(* PLC project services, CODESYS STW CODESYS V3.5 SP11 - ESX-3CS *)
(* stored: creationDateTime 2026-05-19T11:35:05.3616724, version 0.1, modificationDateTime 2026-02-03T11:13:35, organization Isoloader *)

TYPE t_bms_charge_state : (cBMSChargeStateShutdown := 0, cBMSChargeStateDC := 1, cBMSChargeStateAC := 2, cBMSChargeStateOther := 3);
END_TYPE

TYPE t_bms_fault_level : (cBMSFaultLevelNone := 0, cBMSFaultLevelLow := 1, cBMSFaultLevelMedium := 2, cBMSFaultLevelSevere := 3);
END_TYPE

TYPE t_bms_state : (cBMSStateShutdown := 0, cBMSStateStandby := 1, cBMSStateDisconnected := 2, cBMSStateConnected := 3);
END_TYPE

TYPE t_tms_state : (cTMSStateShutdown := 0, cTMSStateCooling := 1, cTMSStateHeating := 2, cTMSStateCirculation := 3);
END_TYPE

TYPE t_charger_diagnostic : (cChargingDiagnostic := 0, cChargingDiagnosticNotOperational := 1, cChargingDiagnosticDisconnected := 2, cChargingDiagnosticConnectedError := 3, cChargingDiagnosticConnectedStandby := 4, cChargingDiagnosticNotInChargingState := 5, cChargingDiagnosticTargetSOCReached := 6, cChargingDiagnosticBMSShutdown := 7, cChargingDiagnosticConnected := 8, cChargingDiagnosticConnectedCharging := 9);
END_TYPE

TYPE t_obc_state : (cOBCStateDisconnected := 0, cOBCStateCharging := 1, cOBCStateStandby := 2, cOBCStateError := 3);
END_TYPE

TYPE t_obc_status : (cOBCStatusNone := 0, cOBCStatusCharging := 1, cOBCStatusStandby := 2, cOBCStatusError := 3);
END_TYPE

TYPE t_active_state : (cActiveStateNone := 0, cActiveStatePre := 1, cActiveStatePost := 2, cActiveStateActive := 3);
END_TYPE

TYPE t_adjust_state : (cAdjustStateNone := 0, cAdjustStateGood := 1, cAdjustStateAdjusting := 2, cAdjustStateError := 3);
END_TYPE

(* {attribute 'qualified_only'} *)
TYPE t_channel_state : (cChannelStateNone := 0, cChannelStateError := 1, cChannelStateOverflow := 2, cChannelStateHeartbeat := 3, cChannelStateEmergency := 4, cChannelStateStarting := 5, cChannelStateReady := 6, cChannelStateGood := 7);
END_TYPE

(* {attribute 'qualified_only'} *)
TYPE t_controller_status : (cControllerStatusNone := 0, cControllerStatusFault := 1, cControllerStatusNotReady := 2, cControllerStatusOnline := 3, cControllerStatusWarning := 4, cControllerStatusReady := 5, cControllerStatusOperating := 6);
END_TYPE

TYPE t_data_type : (cDataTypeNone := 0, cDataTypeEnum := 1, cDataTypeString := 2, cDataTypeUSINT := 3, cDataTypeUINT := 4, cDataTypeULINT := 5, cDataTypeUDINT := 6, cDataTypeINT := 7, cDataTypePercentage := 8, cDataTypeReal := 9, cDataTypeDWORD := 10, cDataTypeBool := 11);
END_TYPE

TYPE t_debug_mask : (cDebugNone := 16#0, cDebugWaitForLog := 16#1, cDebugEnableFailSafeOnCrash := 16#2, cDebugDisableWatchdog := 16#4, cDebugSimulateCrash := 16#100, cDebugSimulateA := 16#200, cDebugSimulateB := 16#400, cDebugSimulateC := 16#800);
END_TYPE

TYPE t_enum_type : (cEnumTypeNone := 0, cEnumTypeActiveState := 1, cEnumTypeAdjustState := 2, cEnumTypeChannelState := 3, cEnumTypeControllerStatus := 4, cEnumTypeDebugMask := 5, cEnumTypeEventCode := 6, cEnumTypeFunctionalMode := 7, cEnumTypeInputMode := 8, cEnumTypeInterlockState := 9, cEnumTypeLedCode := 10, cEnumTypeLockState := 11, cEnumTypeOperatingMethod := 12, cEnumTypeProgMovCode := 13, cEnumTypeProgMovState := 14, cEnumTypeReadyState := 15, cEnumTypeRunState := 16, cEnumTypeShutdownCode := 17, cEnumTypeSpreaderExtensionMethod := 18, cEnumTypeSpreaderExtensionState := 19, cEnumTypeStateCode := 20, cEnumTypeSteerMode := 21, cEnumTypeSubsystem := 22, cEnumTypeSystemMethod := 23, cEnumTypeSystemState := 24, cEnumTypeTopbeamsState := 25, cEnumTypeUiEventCode := 26, cEnumTypeUiId := 27, cEnumTypeUiMode := 28, cEnumTypeUiOrientation := 29, cEnumTypeBMSChargeState := 30, cEnumTypeBMSFaultLevel := 31, cEnumTypeBMSState := 32, cEnumTypeChannelMask := 33, cEnumTypeOBCState := 34, cEnumTypeOBCStatus := 35, cEnumTypeTMSState := 36, cEnumTypeTokenType := 37, cEnumTypeSystemControl := 38, cEnumTypeSeverity := 39, cEnumTypeChargeQualifier := 40, cEnumTypeExecuteOption := 41, cEnumTypeExecuteReturn := 42, cEnumTypeValueStyle := 43, cEnumTypeDataType := 44);
END_TYPE

TYPE t_event_code : (cECNone := 0, cECSystemControl := 1, cECAllowUpState := 2, cECAllowDownState := 3, cECForceMaxState := 4, cECNextState := 5, cECModulation := 6, cECChargeModulation := 8, cECMovementInputInterlock := 9, cECMovementChargeInterlock := 10, cECSecondaryPowerModulation := 11, cECTransitionInitializedStandby := 12, cECTransitionStandbyPreparing := 13, cECTransitionStandbyInitialized := 14, cECTransitionPreparingPreOperational := 15, cECTransitionPreparingCharging := 16, cECTransitionPreparingStandby := 17, cECTransitionChargingPreparing := 18, cECTransitionPreOperationalPreparing := 19, cECTransitionPoweringUpGoOperational := 20, cECTransitionGoOperationalOperational := 21, cECTransitionExitOperationalPoweringDown := 22, cECTransitionPoweringDownPreOperational := 23, cECMetric := 24, cECMax := 63);
END_TYPE

(* {attribute 'qualified_only'} *)
TYPE t_functional_mode : (cFunctionalModeAny := 0, cFunctionalModeDefault := 1, cFunctionalModeTravel := 2, cFunctionalModeLift := 3, cFunctionalModeSpreaderConfiguration := 4, cFunctionalModeTopbeamConfiguration := 5);
END_TYPE

(* {attribute 'qualified_only'} *)
TYPE t_input_mode : (cInputModeNone := 0, cInputModeDefault := 1, cInputModeSpreaderConfiguration := 2, cInputModeTopbeamConfiguration := 3);
END_TYPE

TYPE t_interlock_state : (cInterlockStateNone := 0, cInterlockStateFailure := 1, cInterlockStateError := 2, cInterlockStateErrorNegative := 3, cInterlockStateErrorPositive := 4, cInterlockStateWarning := 5, cInterlockStateOveride := 6, cInterlockStateGood := 7);
END_TYPE

TYPE t_led_code : (cLEDCodeNone := 0, cLEDCodeStartup := 1, cLEDCodeStandby := 2, cLEDCodeNormal := 3, cLEDCodeMaintenance := 4, cLEDCodeSoftwareCrash := 5, cLEDCodeWatchDogDisabled := 6, cLEDCodeFailSafe := 7, cLEDCodeFailSafeSevere := 8);
END_TYPE

(* {attribute 'qualified_only'} *)
TYPE t_lock_state : (cLockStateNone := 0, cLockStateUnlocked := 1, cLockStateLocked := 2, cLockStatePartial := 3);
END_TYPE

(* values of t_machine_state_id: cMSIdSystemState: operating state; cMSIdLocalMessageText: local UIState *)

{attribute 'qualified_only'}
{attribute 'strict'}
TYPE t_machine_state_id : (cMSIdNone := 0, cMSIdSystemState := 1, cMSIdSystemMethodRequest := 2, cMSIdOperatingMode := 3, cMSIdOperatingModeRequest := 4, cMSIdRadioModeResponse := 5, cMSIdMachineHours := 6, cMSIdLightsStatus := 12, cMSIdToggleLightsRequest := 13, cMSIdSpeedModeSlow := 14, cMSIdToggleSpeedModeRequest := 15, cMSIdBatteryLevel := 20, cMSIdMainCurrent := 21, cMSIdChargingCurrent := 22, cMSIdEngineState := 23, cMSIdSteerModeStatus := 30, cMSIdSteerModeRequest := 31, cMSIdSteerModeRequest2WS := 32, cMSIdSteerModeRequest4WS := 33, cMSIdSteerModeRequest4WS90 := 34, cMSIdSteerModeRequestLateral := 35, cMSIdSteerModeRequestCarousel := 36, cMSIdSteerStateA := 37, cMSIdSteerStateB := 38, cMSIdSteerStateC := 39, cMSIdSteerStateD := 40, cMSIdTravelVelocity := 41, cMSIdTravelInterlock := 42, cMSIdTravelInterlockTrace := 43, cMSIdTopbeamABPosition := 44, cMSIdTopbeamCDPosition := 45, cMSIdTopbeamABInterlock := 46, cMSIdTopbeamCDInterlock := 47, cMSIdTopbeamABInterlockTrace := 48, cMSIdTopbeamCDInterlockTrace := 49, cMSIdLiftABPosition := 50, cMSIdLiftCDPosition := 51, cMSIdLiftABInterlock := 52, cMSIdLiftCDInterlock := 53, cMSIdLiftABInterlockTrace := 54, cMSIdLiftCDInterlockTrace := 55, cMSIdLiftTopRequest := 56, cMSIdSpreaderGrabArms := 60, cMSIdToggleSpreaderGrabArmsRequest := 61, cMSIdSpreaderTelescopingExtensionStateRequest6m := 62, cMSIdSpreaderTelescopingExtensionStateRequest9m := 63, cMSIdSpreaderTelescopingExtensionStateRequest12m := 64, cMSIDSpreaderState := 65, cMSIDSpreaderStateA := 66, cMSIDSpreaderStateB := 67, cMSIDSpreaderStateC := 68, cMSIDSpreaderStateD := 69, cMSIDSpreaderLowered := 70, cMSIDSpreaderLoweredA := 71, cMSIDSpreaderLoweredB := 72, cMSIDSpreaderLoweredC := 73, cMSIDSpreaderLoweredD := 74, cMSIdSpreaderTelescopingControl := 75, cMSIdSpreaderGrabArmsDeployControl := 76, cMSIdSpreaderGrabArmsExtendABRequest := 77, cMSIdSpreaderGrabArmsRetractABRequest := 78, cMSIdSpreaderGrabArmsExtendCDRequest := 79, cMSIdSpreaderGrabArmsRetractCDRequest := 80, cMSIdConfigureState := 85, cMSIdConfigureStateValid := 86, cMSIdConfigureMethodRequest := 87, cMSIdReconfigureCheckingRequest := 88, cMSIdUnloadedState := 89, cMSIdLevelState := 90, cMSIdMastsState := 91, cMSIdReconfigureMastsRequest := 92, cMSIdTopbeamsState := 93, cMSIdReconfigureTopbeamsRequest := 94, cMSIdMastAThrottle := 100, cMSIdMastBThrottle := 101, cMSIdMastCThrottle := 102, cMSIdMastDThrottle := 103, cMSIdTopbeamABThrottle := 104, cMSIdTopbeamCDThrottle := 105, cMSIdLocalMessageText := 110, cMSIdLocalMessageDisplayCode := 111, cMSIdLocalStatusText := 112, cMSIdLocalStatusDisplayCode := 113, cMSIdLocalButtonSteerModeSelectEnter := 115, cMSIdLocalButtonSteerModeSelectSwitch := 116, cMSIdLocalButtonSteerModeSelectExit := 117, cMSIDLocalAckMessageEnter := 118, cMSIDLocalAckMessageExit := 119, cMSIDLocalFlashMessageEnter := 120, cMSIDLocalFlashMessageExit := 121, cMSIdLocalButtonConfigureEnter := 122, cMSIdLocalButtonConfigureSwitch := 123, cMSIdLocalButtonConfigureExit := 124, cMSIdLocalButtonMastsSelectEnter := 125, cMSIdLocalButtonMastsSelectSwitch := 126, cMSIdLocalButtonMastsSelectExit := 127, cMSIdLocalButtonTopbeamsSelectEnter := 128, cMSIdLocalButtonTopbeamsSelectSwitch := 129, cMSIdLocalButtonTopbeamsSelectExit := 130, cMSIdLocalButtonUnloadedSelectEnter := 131, cMSIdLocalButtonUnloadedSelectSwitch := 132, cMSIdLocalButtonUnloadedSelectExit := 133, cMSIdLocalButtonLevelSelectEnter := 134, cMSIdLocalButtonLevelSelectSwitch := 135, cMSIdLocalButtonLevelSelectExit := 136, cMSIdLocalButtonSpreaderDeployControlEnter := 137, cMSIdLocalButtonSpreaderDeployControlExit := 138, cMSIdLocalDiagnosticsMode := 141, cMSIdLocalToggleDiagnosticsMode := 142, cMSIdTopbeamConfigurationEnabled := 143, cMSIdMax := 144);
END_TYPE

(* /{attribute 'qualified_only'} *)
TYPE t_operating_method : (cOperatingMethodNone := 0, cOperatingMethodPark := 1, cOperatingMethodUnpark := 2, cOperatingMethodLock := 3, cOperatingMethodLockWithoutPark := 4, cOperatingMethodUnlock := 5, cOperatingMethodSlow := 6, cOperatingMethodNormal := 7);
END_TYPE

(* {attribute 'qualified_only'} *)
TYPE t_operating_mode : (cOperatingModeInoperable := 0, cOperatingModeParked := 1, cOperatingModeParking := 2, cOperatingModeLocked := 3, cOperatingModeUnparking := 4, cOperatingModeStopped := 5, cOperatingModeStalled := 6, cOperatingModeSlow := 7, cOperatingModeNormal := 8);
END_TYPE

TYPE t_prog_mov_code : (cProgMovCodeNone := 0, cProgMovCode_Lift_Top := 1, cProgMovCode_Lift_Bottom := 2, cProgMovCode_Lift_StandardOnGround := 3, cProgMovCode_Lift_StandardGround := 4, cProgMovCode_Lift_StandardTruck := 5, cProgMovCode_Lift_StandardStack1 := 6, cProgMovCode_Lift_StandardStack2 := 7, cProgMovCode_Lift_HicubeOnGround := 8, cProgMovCode_Lift_HicubeGround := 9, cProgMovCode_Lift_HicubeTruck := 10, cProgMovCode_Lift_HicubeStack1 := 11, cProgMovCode_Lift_HicubeStack2 := 12, cProgMovCode_Travel_LAT0_Forward := 20, cProgMovCode_Travel_LAT0_Reverse := 21, cProgMovCode_Travel_LAT0_4WS_Forward := 22, cProgMovCode_Travel_LAT0_4WS_Reverse := 23, cProgMovCode_Travel_LATPos90_Forward := 24, cProgMovCode_Travel_LATPos90_Reverse := 25, cProgMovCode_Travel_LATNeg90_Forward := 26, cProgMovCode_Travel_LATNeg90_Reverse := 27, cProgMovCode_Test1 := 28, cProgMovCode_Test2 := 29, cProgMovCode_Steer_0 := 30, cProgMovCode_Clear := 31);
END_TYPE

TYPE t_prog_mov_state : (cProgMovStateDisabled := 0, cProgMovStateInactive := 1, cProgMovStatePreparing := 2, cProgMovStateWaiting := 3, cProgMovStateRunning := 4, cProgMovStateFinishing := 5, cProgMovStateLeaving := 6);
END_TYPE

(* {attribute 'qualified_only'} *)
TYPE t_ready_state : (cReadyStateNone := 0, cReadyStateNotReady := 1, cReadyStatePartial := 2, cReadyStateReady := 3);
END_TYPE

TYPE t_run_state : (cRunStateNone := 0, cRunStateStart := 1, cRunStateStop := 2);
END_TYPE

(* {attribute 'qualified_only'} *)
TYPE t_shutdown_code : (cShutdownCodeUnknown := 0, cShutdownCodeIgnition := 1, cShutdownCodeSoftware := 2, cShutdownCodeSupervisor := 3, cShutdownCodeCrashDetected := 4, cShutdownCodeTrapDetected := 5);
END_TYPE

TYPE t_spreader_extension_method : (cSpreaderExtensionMethodNone := 0, cSpreaderExtensionMethodABExtend := 1, cSpreaderExtensionMethodCDExtend := 2, cSpreaderExtensionMethodABRetract := 3, cSpreaderExtensionMethodCDRetract := 4);
END_TYPE

TYPE t_spreader_extension_state : (cSpreaderExtensionStateNone := 0, cSpreaderExtensionState6m := 1, cSpreaderExtensionState9m := 2, cSpreaderExtensionState12m := 3);
END_TYPE

(* values of t_state_code: cACBMSChargeStateMismatch: cACBMSStateMismatch := 32,; cDCNone: 87 *)

TYPE t_state_code : (cSCNone := 0, cACSteerALargeSensorDelta := 1, cACSecondaryNotRunning := 2, cACSecondaryWaiting := 3, cACSecondaryNotRunningModulation := 4, cACSecondaryRunStateMismatch := 35, cACSecondaryTemperature := 39, cACChannelNotGood := 5, cACChannelOperationalFail := 66, cACChannelNotOperational := 6, cACChannelOverflow := 7, cACChannelSlaveFailed := 8, cACCANOpenSlaveNotOperational := 9, cACCANOpenSlaveModulation := 43, cACCANOpenSlaveAllowableUp := 44, cACCANOpenMasterNotOperational := 62, cACCANOpenMasterModulation := 63, cACCANOpenMasterAllowableUp := 64, cACCANOpenSlaveNoValidTransmissions := 49, cACCANOpenSlaveNotify := 36, cACCANOpenSlaveBlock := 37, cACCANOpenSlaveStop := 38, cACUInterfaceEstop := 10, cACUInterfaceStop := 11, cACUInterfaceEmgy := 12, cACUInterfaceNotReady := 13, cACControllerTemperatureCutback := 14, cACMotorTemperatureCutback := 15, cACMotorTemperatureSensor := 73, cACCoolantReservoir := 16, cACCoolantTempHotCutback := 17, cACCoolantTempColdCutback := 18, cACCoolantHeating := 19, cACCoolantChilling := 20, cACCoolantSecondaryPowerFailHeatingCooling := 45, cACCoolantSecondaryPowerFailPump := 46, cACChargerOBCError := 21, cACBMSAvailabilityInsufficient := 22, cACBMSAvailabilityLimited := 48, cBMSChargeAvailabilityLimited := 51, cBMSChargeAvailabilityLimitedSevere := 52, cBMSDischargeAvailabilityLimited := 53, cBMSDischargeAvailabilityLimitedSevere := 54, cACSOCBelowOperatingMinimum := 23, cACSOCBelowStandbyMinimum := 24, cACSOCWarningLow := 47, cACBMSNotConnected := 25, cACBMSFailToConnect := 32, cACBMSChargeCutback := 26, cACBMSDischargeCutback := 27, cACBMSRequestDisconnect := 50, cACBMSFault := 55, cACBackupBatteryVoltageLow := 28, cACBeaconsSecondaryPowerFail := 29, cACSecondaryPowerFail := 30, cACTMSStateMismatch := 31, cACBMSChargeStateMismatch := 33, cACBMSSOCMismatch := 70, cACBMSVoltageMismatch := 71, cACBMSCurrentMismatch := 72, cACSensorRangeError := 34, cACHydraulicFilter := 56, cACHydraulicTemperature := 57, cACBrakeLowHydraulicPressure := 58, cACOutputFailure := 59, cACDeviceTemperature := 60, cACDeviceVoltage := 61, cACSoftwareCrash := 65, cACFailSafeMode := 67, cACMaintenanceMode := 68, cACWatchdogDisabled := 69, cACExecutionFailed := 74, cACPersistedCommands := 86, cACSoftware := 75, cACConfiguration := 76, cACVoltage := 77, cACTemperature := 78, cACRelayFuse := 79, cACFuse := 80, cACSubsystem := 81, cACConsumable := 82, cACHeartbeat := 83, cACOutput := 84, cACControlSignal := 85, cDCNone := (128 + 0), cDCChargerStandby := (128 + 1), cDCChargerConnected := (128 + 2), cDCChargerDisconnected := (128 + 3), cDCTMSCooling := (128 + 4), cDCTMSHeating := (128 + 5), cDCBMSTMSCooling := (128 + 6), cDCBMSTMSHeating := (128 + 7), cDCBMSTMSNoCirculation := (128 + 8), cDCNonexx := (128 + 10), cCCNone := (192 + 0), cCCChargerStandby := (192 + 1), cCCChargerConnected := (192 + 2), cCCChargerDisconnected := (192 + 3), cCCWaitingForBrakeDisengaged := (192 + 5), cCCWaitingForParked := (192 + 6), cCCCommandStart := (192 + 7), cCCCommandStop := (192 + 8), cCCStopOnTimeout := (192 + 9), cCCLockoutInterlock := (192 + 10), cCCPosOnlyInterlock := (192 + 11), cCCScaledInterlock := (192 + 12), cCCThresholdInterlock := (192 + 13), cCCSynchronousInterlock := (192 + 14), cCCTwistlocksReadyInterlock := (192 + 15), cCCAutomaticStart := (192 + 16), cCCSyncState := (192 + 17), cCCCurrentUserNotEnabled := (192 + 18), cCCStandby := (192 + 19), cCCCycleOutput := (192 + 20), cSCMax := 254);
END_TYPE

(* {attribute 'qualified_only'} *)
TYPE t_steer_mode : (cSteerModeNone := 0, cSteerMode4WS := 1, cSteerModeLateral := 2, cSteerModeCarousel := 3, cSteerModeReconfigure := 4, cSteerModeLateralNeg90 := 5, cSteerModeLateralPos90 := 6, cSteerModeCustom := 7);
END_TYPE

(* values of t_subsystem: cSubsystemSideshiftAB: foobar; cSubsystemSpreaderPowerPack: foobar; cSubsystemTwistlockA: foobar *)

TYPE t_subsystem : (cSubsystemNone := 0, cSubsystemSpreader := 1, cSubsystemBeacons := 2, cSubsystemCabin := 3, cSubsystemLights := 4, cSubsystemPowerpack := 5, cSubsystemSideshiftAB := 6, cSubsystemSideshiftCD := 7, cSubsystemSpreaderPowerPack := 8, cSubsystemSteerA := 9, cSubsystemSteerB := 10, cSubsystemSteerC := 11, cSubsystemSteerD := 12, cSubsystemTravelA := 13, cSubsystemTravelB := 14, cSubsystemTravelC := 15, cSubsystemTravelD := 16, cSubsystemWinchA := 17, cSubsystemWinchB := 18, cSubsystemWinchC := 19, cSubsystemWinchD := 20, cSubsystemTwistlockA := 21, cSubsystemTwistlockB := 22, cSubsystemTwistlockC := 23, cSubsystemTwistlockD := 24, cSubsystemTopbeamAB := 25, cSubsystemTopbeamCD := 26, cSubsystemCANBusSystem := 27, cSubsystemCANBusDrive := 28, cSubsystemBattery := 29, cSubsystemSecondary := 30, cSubsystemUInterface := 31, cSubsystemHydraulics := 32, cSubsystemLift := 33, cSubsystemTravel := 34, cSubsystemSteer := 35, cSubsystemMachine := 36, cSubsystemMax := 37);
END_TYPE

(* values of t_system_method: cSystemMethodNone: requests only *)

(* {attribute 'qualified_only'} *)
TYPE t_system_method : (cSystemMethodNone := 0, cSystemMethodStart := 1, cSystemMethodStop := 2, cSystemMethodEStop := 3, cSystemMethodReset := 4);
END_TYPE

(* /{attribute 'qualified_only'} *)
TYPE t_system_state : (cSystemStateNone := 0, cSystemStateInitialized := 1, cSystemStateStandby := 2, cSystemStatePreparing := 3, cSystemStateCharging := 4, cSystemStatePreOperational := 5, cSystemStatePoweringDown := 6, cSystemStatePoweringUp := 7, cSystemStateGoOperational := 8, cSystemStateExitOperational := 9, cSystemStateOperational := 10);
END_TYPE

(* /{attribute 'qualified_only'} *)
TYPE t_topbeams_state : (cTopbeamsStateNone := 0, cTopbeamsStateRetracted := 1, cTopbeamsStateExtended := 2, cTopbeamsStateMiddle := 3);
END_TYPE

TYPE t_ui_event_code : (cUIEventCodeNone := 0, cUIEventCodeToggleLights := 1, cUIEventCodeUIModeResponse := 2, cUIEventCodeToggleSpreaderConfiguration := 3, cUIEventCodeSpreaderExtensionAutoCommand := 4, cUIEventCodeSpreaderRetractionAutoCommand := 5, cUIEventCodeInitiate := 7, cUIEventCodeStart := 8, cUIEventCodeStop := 9, cUIEventCodeProgMovStart := 10, cUIEventCodeProgMovMax := 31);
END_TYPE

TYPE t_ui_id : (cUIIdNone := 0, cUIIdA := 1, cUIIdB := 2);
END_TYPE

(* {attribute 'qualified_only'} *)
TYPE t_ui_mode : (cUIModeInoperable := 0, cUIModeSlave := 1, cUIModeMaster := 2, cUIModeSingle := 3);
END_TYPE

(* {attribute 'qualified_only'} *)
TYPE t_ui_orientation : (cUIOrientationNone := 0, cUIOrientationForward := 1, cUIOrientationSide := 2, cUIOrientationReverse := 3, cUIOrientationOpposite := 4);
END_TYPE

TYPE t_value_style : (cValueStyleConfigurable := 0, cValueStyleParameter := 1, cValueStyleTrigger := 2);
END_TYPE

TYPE t_charge_interlock : ReportableContextChargeModulationRCSM;
END_TYPE

TYPE t_movement_interlock : MovementInterlock;
END_TYPE

TYPE t_metric : Metric;
END_TYPE

TYPE t_metric_ptr : POINTER TO t_metric;
END_TYPE

TYPE t_metric_set : ARRAY[1..8] OF t_metric_ptr;
END_TYPE

TYPE t_packer : Packer;
END_TYPE

TYPE t_packer_ptr : POINTER TO Packer;
END_TYPE

TYPE t_packer_set : ARRAY[1..16] OF t_packer_ptr;
END_TYPE

TYPE t_bitarray : ARRAY[1..64] OF BOOL;
END_TYPE

TYPE t_packet : PacketCANBus;
END_TYPE

TYPE t_timestep : UDINT;
END_TYPE

TYPE t_connection_handler : ConnectionHandler;
END_TYPE

TYPE t_execution_queue_item : STRUCT
  depth : USINT;
  particle : t_particle_ptr;
END_STRUCT;
END_TYPE

TYPE t_socket_state : (cSocketStateInvalid := 0, cSocketStateCreate := 1, cSocketStateIOCtl := 2, cSocketStateBind := 3, cSocketStateListen := 4, cSocketStateConnect := 5, cSocketStateConnected := 6, cSocketStateClose := 7);
END_TYPE

TYPE t_tcp_connection : TCPConnection;
END_TYPE

TYPE t_uinterface_diagnostic : (cUInterfaceDiagnosticOK := 0, cUInterfaceDiagnosticEstop := 1, cUInterfaceDiagnosticStop := 2, cUInterfaceDiagnosticEmgy := 3, cUInterfaceDiagnosticTimedStop := 4, cUInterfaceDiagnosticNotReady := 5, cUInterfaceDiagnosticInoperable := 6, cUInterfaceDiagnosticNotMaster := 7);
END_TYPE

TYPE t_argument : STRUCT
  parameter : t_token_type;
  value : t_token_string;
  processed : BOOL;
END_STRUCT;
END_TYPE

TYPE t_arguments_list : ARRAY[1..cExecuteArgumentListCount] OF t_argument;
END_TYPE

TYPE t_command_definition : STRUCT
  command : t_token_type;
  options : t_options_list;
  optionCount : USINT;
  pairMinCount : USINT;
  pairMaxCount : USINT;
  readwrite : BOOL;
  description : REFERENCE TO t_medium_string;
END_STRUCT;
END_TYPE

TYPE t_command_request : STRUCT
  particle : POINTER TO t_particle;
  command : t_token_type;
  options : t_options_list;
  optionCount : USINT;
  arguments : t_arguments_list;
  argumentCount : USINT;
END_STRUCT;
END_TYPE

TYPE t_command_store : STRUCT
  particle : t_particle_id;
  command : t_token_type;
  options : t_options_list;
  optionCount : USINT;
  arguments : t_arguments_list;
  argumentCount : USINT;
END_STRUCT;
END_TYPE

TYPE t_execute_option : (cExecuteOptionNone := 0, cExecuteOptionRecurse := 1, cExecuteOptionVerbose := 2, cExecuteOptionParameter := 3, cExecuteOptionSyntax := 4, cExecuteOptionChildren := 5, cExecuteOptionExecutor := 6, cExecuteOptionSubsystems := 7, cExecuteOptionPersist := 8, cExecuteOptionAll := 9, cExecuteOptionMetadata := 10);
END_TYPE

TYPE t_execute_return : (cExecuteReturnOK := 0, cExecuteReturnUnknownArgumentValue := 1, cExecuteReturnUnsupportedForParticleType := 2, cExecuteReturnNullParticle := 3, cExecuteReturnSetOverflow := 4, cExecuteReturnUnknownOption := 5, cExecuteReturnOKNOK := 6, cExecuteReturnUnknownCommand := 7, cExecuteReturnUnknownParameter := 8, cExecuteReturnUnsupportedRecurse := 9, cExecuteReturnExecutionQueueOverflow := 10, cExecuteReturnExecutionQueueNullParticle := 11, cExecuteReturnParseParameterError := 12, cExecuteReturnUnknownOptionChannelMask := 13, cExecuteReturnUnknownOptionDebugMask := 14, cExecuteReturnIllegalIndex := 15, cExecuteReturnMissingArgument := 16, cExecuteReturnTooFewArguments := 17, cExecuteReturnTooManyArguments := 18, cExecuteReturnInternalError := 19, cExecuteReturnPersistFailed := 20, cExecuteReturnUnprocessedArguments := 21, cExecuteReturnExecutionExecutorFailed := 22, cExecuteReturnExecutionSyntax := 23, cExecuteReturnExecutionSyntaxIncompleteRequest := 24, cExecuteReturnExecutionSyntaxIncompleteParameter := 25, cExecuteReturnExecutionSyntaxIncompleteName := 26, cExecuteReturnExecutionSyntaxTokenOverflow := 27, cExecuteReturnExecutionSyntaxStartWithName := 28, cExecuteReturnExecutionSyntaxCommandAfterName := 29, cExecuteReturnExecutionSyntaxDuplicateCommands := 30, cExecuteReturnExecutionSyntaxUnkownName := 31, cExecuteReturnExecutionSyntaxUnkownNameForParameter := 32, cExecuteReturnExecutionSyntaxTooManyOptions := 33, cExecuteReturnExecutionSyntaxUnbounded := 34, cExecuteReturnReadOnly := 35);
END_TYPE

TYPE t_execute_source : ExecuteSource;
END_TYPE

TYPE t_fqtoken_string : STRING(128);
END_TYPE

TYPE t_name : t_medium_string;
END_TYPE

TYPE t_options_list : ARRAY[1..cExecuteOptionListCount] OF t_execute_option;
END_TYPE

TYPE t_parse_token_type : (cParseTokenNone := 0, cParseTokenOverflow := 1, cParseTokenError := 2, cParseTokenSimple := 3, cParseTokenName := 4, cParseTokenParameter := 5, cParseTokenOption := 6, cParseTokenTerminator := 7, cParseTokenFinished := 8);
END_TYPE

TYPE t_particle : Particle;
END_TYPE

TYPE t_particle_id : UINT;
END_TYPE

TYPE t_particle_nop : NonOperationalParticleSet;
END_TYPE

TYPE t_particle_op : OperationalParticleSet;
END_TYPE

TYPE t_particle_ptr : POINTER TO t_particle;
END_TYPE

TYPE t_token_string : t_medium_string;
END_TYPE

TYPE t_token_string_set : ARRAY[1..cTokenStringSetCount] OF t_token_string;
END_TYPE

TYPE t_token_type : (cTokenNone := 0, cTokenDescribe := 1, cTokenSyntax := 2, cTokenVerify := 3, cTokenIdentify := 4, cTokenRegister := 5, cTokenConfigure := 6, cTokenSetFailSafeMode := 7, cTokenClearFailSafeMode := 8, cTokenFailSafeConfig := 9, cTokenProceed := 10, cTokenList := 11, cTokenDebugMaskAdd := 12, cTokenDebugMaskDelete := 13, cTokenDebugMaskClear := 14, cTokenClose := 15, cTokenExport := 16, cTokenClear := 17, cTokenDeregister := 18, cTokenTrigger := 19, cTokenChannelMaskAdd := 20, cTokenChannelMaskDelete := 21, cTokenChannelMaskClear := 22, cTokenChannelIndex := 23, cTokenValue := 24, cTokenOverrideValue := 25, cTokenOverride := 26, cTokenValueType := 27, cTokenMeaning := 28, cTokenOverrideMeaning := 29, cTokenRawIndex := 30, cTokenIndex := 31, cTokenUnknown := 32, cTokenObject := 33, cTokenFeature := 34, cTokenZero := 35, sTokenUpper := 36, sTokenExecute := 37, cTokenThreshold := 38, cTokenHysteresis := 39, cTokenImport := 40);
END_TYPE

TYPE t_summary_lines : ARRAY[1..cSummaryLines] OF t_long_string;
END_TYPE

TYPE t_channel : ReportableChannel;
END_TYPE

TYPE t_channel_id : (cReportableChannelDefault := 1);
END_TYPE

TYPE t_channel_manager : ReportableChannelManager;
END_TYPE

TYPE t_channel_mask : (cChannelNone := 16#0, cChannelUIRadio := 16#1, cChannelUICabin := 16#2, cChannelLogTCP := 16#4, cChannelUIRCache := 16#8, cChannelMaster := 16#10, cChannelEdgeLog := 16#20, cChannelEdgeStateMetric := 16#40, cChannelEdgeValueMetric := 16#80, cChannelEdgeTrace := 16#100);
END_TYPE

TYPE t_channel_set : ARRAY[1..8] OF POINTER TO t_channel;
END_TYPE

TYPE t_charge_qualifier : (cChargeQualifierBoth := 0, cChargeQualifierCharge := 1, cChargeQualifierDischarge := 2, cChargeQualifierNone := 3);
END_TYPE

TYPE t_diagnostic_code : (xDCNone := 0, xDCChargerStandby := 1, xDCChargerConnected := 2, xDCChargerDisconnected := 3, xDCNonexx := 10);
END_TYPE

TYPE t_reportable : Reportable;
END_TYPE

TYPE t_reportable_array : ARRAY[1..16] OF POINTER TO t_reportable;
END_TYPE

TYPE t_reportable_set : ReportableSet;
END_TYPE

TYPE t_reportableevent : ReportableEvent;
END_TYPE

TYPE t_reportablestate : ReportableState;
END_TYPE

TYPE t_severity : (cSeverityNone := 0, cSeverityWarning := 1, cSeverityError := 2, cSeverityCritical := 3);
END_TYPE

TYPE t_state_context : LWORD;
END_TYPE

TYPE t_stream : Stream;
END_TYPE

TYPE t_stream_string : STRING;
END_TYPE

TYPE t_system_control : (cSystemControlReset := 0, cSystemControlEStop := 1, cSystemControlStop := 2, cSystemControlStart := 3, cSystemControlNone := 4);
END_TYPE

TYPE t_ui_reportable : STRUCT
  valid : BOOL;
  state : t_state_code;
  event : t_event_code;
  subsystem : t_subsystem;
  active : BOOL;
END_STRUCT;
END_TYPE

{attribute 'enable_dynamic_creation'}
TYPE t_enum_option_definition : STRUCT
  option : INT;
  token : t_token_string;
  description : t_long_string;
END_STRUCT;
END_TYPE

VAR_GLOBAL CONSTANT  (* GlobalVariablesServices *)
  cSummaryLines : USINT := 8;
  cExecuteOptionListCount : USINT := 8;
  cExecuteArgumentListCount : USINT := 4;
  cTokenStringSetCount : USINT := 16;
  sDefaultIdentity : t_long_string := 'Particle';
  sDefaultName : t_name := 'Particle';
  sParticle : t_medium_string := 'Particle';
  gNameSpace : t_token_string;
  gParticleDebugIdA : t_particle_id := 0;
  gParticleDebugIdB : t_particle_id := 0;
  gTypeHandler : GlobalTypeHandler;
  gSystemServices : REFERENCE TO System;
  gDebugFlags : t_persistent_uint;
  gStateCodeLastUnknown : t_state_code;
  gEventCodeLastUnknown : t_event_code;
  sLastParticleId : t_particle_id := 0;
  sCommandConfigure : t_command_definition := (command := cTokenConfigure, options := [cExecuteOptionRecurse, cExecuteOptionSubsystems], optionCount := 2, pairMinCount := 1, pairMaxCount := 4);
  sCommandVerify : t_command_definition := (command := cTokenVerify, options := [cExecuteOptionRecurse, cExecuteOptionSubsystems], optionCount := 2);
  sCommandSetFailSafeMode : t_command_definition := (command := cTokenSetFailSafeMode);
  sCommandClearFailSafeMode : t_command_definition := (command := cTokenClearFailSafeMode);
  sCommandDescribe : t_command_definition := (command := cTokenDescribe, options := [cExecuteOptionVerbose, cExecuteOptionParameter, cExecuteOptionRecurse, cExecuteOptionSyntax, cExecuteOptionChildren, cExecuteOptionExecutor, cExecuteOptionSubsystems, cExecuteOptionMetadata], optionCount := 8);
  sCommandIdentify : t_command_definition := (command := cTokenIdentify, options := [cExecuteOptionRecurse, cExecuteOptionExecutor, cExecuteOptionSubsystems], optionCount := 3);
  sCommandChannelMaskAdd : t_command_definition := (command := cTokenChannelMaskAdd, pairMinCount := 1, pairMaxCount := 1);
  sCommandChannelMaskDelete : t_command_definition := (command := cTokenChannelMaskDelete, pairMinCount := 1, pairMaxCount := 1);
  sCommandChannelMaskClear : t_command_definition := (command := cTokenChannelMaskClear);
  sCommandDebugMaskAdd : t_command_definition := (command := cTokenDebugMaskAdd, pairMinCount := 1, pairMaxCount := 1);
  sCommandDebugMaskDelete : t_command_definition := (command := cTokenDebugMaskDelete, pairMinCount := 1, pairMaxCount := 1);
  sCommandDebugMaskClear : t_command_definition := (command := cTokenDebugMaskClear);
  sCommandExport : t_command_definition := (command := cTokenExport);
  sCommandClear : t_command_definition := (command := cTokenClear, options := [cExecuteOptionAll], optionCount := 1, pairMinCount := 0, pairMaxCount := 1);  (* 'Persistent 4-byte block at given index' *)
  sCommandExecute : t_command_definition := (command := sTokenExecute, options := [cExecuteOptionAll], optionCount := 1, pairMinCount := 0, pairMaxCount := 1);
  sCommandRegister : t_command_definition := (command := cTokenRegister, pairMinCount := 1, pairMaxCount := 1);
  sCommandDeregister : t_command_definition := (command := cTokenDeregister, pairMinCount := 1, pairMaxCount := 1);
  sCommandTrigger : t_command_definition := (command := cTokenTrigger);
  sCommandClose : t_command_definition := (command := cTokenClose);
END_VAR

VAR_GLOBAL  (* GVLallocate *)
  _defaultLongString : t_long_string := 'unallocated';
  _countLongString : UINT := 0;
  _defaultMediumString : t_medium_string := 'unallocated';
  _countMediumString : UINT := 0;
  cDescriptionValue : t_long_string := 'Current value';
  cDescriptionOverrideValue : t_long_string := 'Value if overriden';
  cDescriptionOverride : t_long_string := 'Whether TO override the parameter value';
  cDescriptionThreshold : t_long_string := 'Switching threshold';
  cDescriptionHysteresis : t_long_string := 'Switching hysteresis';
  cDescriptionProceed : t_long_string := 'Parent object is executed';
  cDescriptionFailSafeConfig : t_long_string := 'Parent object is executed when in failsafe mode';
  sTypeHandlerBool : TypeHandlerBool;
  sTypeHandlerDWORD : TypeHandlerDWORD;
  sTypeHandlerPercentage : TypeHandlerPercentage;
  sTypeHandlerREAL : TypeHandlerREAL;
  sTypeHandlerINT : TypeHandlerINT;
  sTypeHandlerUDINT : TypeHandlerUDINT;
  sTypeHandlerUINT : TypeHandlerUINT;
  sTypeHandlerULINT : TypeHandlerULINT;
  sTypeHandlerUSINT : TypeHandlerUSINT;
END_VAR

FUNCTION_BLOCK MovementInterlock EXTENDS ReportableContextSignedModulation
  VAR_INPUT
    lEnableManualTemporaryOveride : BOOL := TRUE;
    lEnableGradualStop : BOOL := FALSE;
  END_VAR
  VAR CONSTANT
    cStopFactor : REAL := 0.89;
    cStopScalingZeroThreshold : REAL := 0.05;
  END_VAR
  VAR
    lStopFactor : REAL := cStopFactor;
    lStopScaling : REAL;
  END_VAR

            ;
          

METHOD operator
                  SUPER^.operator();

IF (InterlockState<=cInterlockStateError) THEN
	IF (lEnableGradualStop) THEN
		lStopScaling := lStopScaling * lStopFactor;
		IF (ABS(lStopScaling)<cStopScalingZeroThreshold) THEN
			lStopScaling := 0.0;			
		END_IF
	ELSE
		lStopScaling := 0.0;
	END_IF
ELSE
	lStopScaling := 1.0;	
END_IF

                
END_METHOD

METHOD stop : t_percentage
  VAR_INPUT
    value : t_percentage;
  END_VAR
                  IF (ABS(value)<cStopScalingZeroThreshold) THEN
	stop := 0.0;
	RETURN;
END_IF

stop := value * lStopScaling;

                
END_METHOD

METHOD update : t_percentage
  VAR_INPUT
    value : t_percentage;
  END_VAR
                  IF ((InterlockState<cInterlockStateOveride) AND
	(gManualTemporaryOveride) AND
	(lEnableManualTemporaryOveride)) THEN
	update := value;
	RETURN;
END_IF

update := SUPER^.update(value);

                
END_METHOD

PROPERTY TypeToken : t_medium_string
GET
                    TypeToken := 'iMovement';
                  
END_GET
END_PROPERTY
END_FUNCTION_BLOCK

FUNCTION_BLOCK TransformIsoscelesTrapezoid
  VAR
    lInRange : BOOL;
    lOffset : t_percentage := 0.0;
    lOuterRegion : t_percentage := 1.0;
    lInnerRegion : t_percentage := 0.95;
    lInnerValue : t_percentage := 1.0;
    lOuterValue : t_percentage := 0.0;
  END_VAR

            
          

METHOD compute : t_percentage
  VAR_INPUT
    input : t_percentage;
  END_VAR
                  input := input - lOffset;

(* range is symmetrical about zero *)
lInRange := (ABS(input)<ABS(lOuterRegion));

(* output or lValue ranges from lInnerValue down to lOuterValue *)
IF (ABS(input)<=ABS(lInnerRegion)) THEN
	compute := lInnerValue;
	RETURN;
END_IF

IF (ABS(input)>=ABS(lOuterRegion)) THEN
	compute := lOuterValue;
	RETURN;
END_IF

IF (ABS(lInnerRegion)=ABS(lOuterRegion)) THEN
	compute := lInnerValue;
	RETURN;
END_IF

(* scale between lInnerValue and lOuterValue - will generally not be signed *)
compute := lInnerValue + (ABS(input)-ABS(lInnerRegion))/(ABS(lOuterRegion)-ABS(lInnerRegion))*(lOuterValue-lInnerValue);


                
END_METHOD

PROPERTY InnerRegion : t_percentage
GET
                    InnerRegion := lInnerRegion;
                  
END_GET
SET
                    lInnerRegion := InnerRegion;
                  
END_SET
END_PROPERTY

PROPERTY InnerValue : t_percentage
GET
                    InnerValue := lInnerValue;
                  
END_GET
SET
                    lInnerValue := InnerValue;
                  
END_SET
END_PROPERTY

PROPERTY InRange : BOOL
GET
                    InRange := lInRange;
                  
END_GET
END_PROPERTY

PROPERTY Offset : t_percentage
GET
                    Offset := lOffset;
                  
END_GET
SET
                    lOffset := Offset;
                  
END_SET
END_PROPERTY

PROPERTY OuterRegion : t_percentage
GET
                    OuterRegion := lOuterRegion;
                  
END_GET
SET
                    lOuterRegion := OuterRegion;
                  
END_SET
END_PROPERTY

PROPERTY OuterValue : t_percentage
GET
                    OuterValue := lOuterValue;
                  
END_GET
SET
                    lOuterValue := OuterValue;
                  
END_SET
END_PROPERTY
END_FUNCTION_BLOCK

FUNCTION_BLOCK CutbackInterlock EXTENDS ReportableChargeModulation
  VAR
    lValue : REAL;
    lInitialCutbackThreshold : REAL;
    lCutoutThreshold : REAL;
    lFactor : REAL;
    lMinimiumThreshold : t_percentage := 0.0;
  END_VAR

            ;
          

METHOD setFactor
                  IF (lCutoutThreshold<=lInitialCutbackThreshold) THEN
	lFactor := 0.0;
ELSE
	lFactor := (-1.0)/(lCutoutThreshold - lInitialCutbackThreshold);
END_IF

                
END_METHOD

METHOD test
  VAR_INPUT
    override : BOOL;
  END_VAR
  VAR
    threshold : t_percentage;
  END_VAR
                  lScalingCharge := 1.0;
lScalingDischarge := 1.0;

IF (lValue>lInitialCutbackThreshold) THEN
	threshold := MAX((1.0 + ((lValue-lInitialCutbackThreshold)*lFactor)),lMinimiumThreshold);
	
	CASE lQualifier OF
		cChargeQualifierBoth:
			lThresholdCharge := threshold;
			lThresholdDischarge := threshold;

		cChargeQualifierCharge:
			lThresholdCharge := threshold;
			lThresholdDischarge := 1.0;
	
		cChargeQualifierDischarge:
			lThresholdCharge := 1.0;
			lThresholdDischarge := threshold;
			
		cChargeQualifierNone:
			lThresholdCharge := 1.0;
			lThresholdDischarge := 1.0;
	END_CASE

	IF ((override) OR
		(lQualifier=cChargeQualifierNone)) THEN
		RETURN;
	END_IF
		
	trigger(FALSE);

	RETURN;
END_IF

lThresholdCharge := 1.0;
lThresholdDischarge := 1.0;

                
END_METHOD

PROPERTY CutoutThreshold : REAL
GET
                    CutoutThreshold := lCutoutThreshold;
                  
END_GET
SET
                    lCutoutThreshold := CutoutThreshold;
setFactor();
                  
END_SET
END_PROPERTY

PROPERTY Factor : REAL
GET
                    Factor := lFactor;
                  
END_GET
END_PROPERTY

PROPERTY InitialCutbackThreshold : REAL
GET
                    InitialCutbackThreshold := lInitialCutbackThreshold;
                  
END_GET
SET
                    lInitialCutbackThreshold := InitialCutbackThreshold;
setFactor();

                  
END_SET
END_PROPERTY

PROPERTY Value : REAL
GET
                    Value := lValue;
                  
END_GET
SET
                    lValue := Value;
                  
END_SET
END_PROPERTY

PROPERTY MinimiumThreshold : t_percentage
GET
                    MinimiumThreshold := lMinimiumThreshold;
                  
END_GET
SET
                    lMinimiumThreshold := MinimiumThreshold;
                  
END_SET
END_PROPERTY
END_FUNCTION_BLOCK

FUNCTION_BLOCK LockoutInterlock EXTENDS ReportableSignedModulation
  VAR
    lValue : BOOL;
  END_VAR

            ;
          

METHOD test
  VAR_INPUT
    override : BOOL;
  END_VAR
                  IF (override) THEN
	RETURN;
END_IF

clear();

IF (lValue) THEN
	lInterlockState:=cInterlockStateError;
	lScalingPositive := 0.0;
	lThresholdPositive := 0.0;
	lScalingNegative := 0.0;
	lThresholdNegative := 0.0;
	
	trigger(FALSE);
END_IF

                
END_METHOD

PROPERTY Value : BOOL
GET
                    Value := lValue;
                  
END_GET
SET
                    lValue := Value;
                  
END_SET
END_PROPERTY
END_FUNCTION_BLOCK

FUNCTION_BLOCK PositiveOnlyInterlock EXTENDS ReportableSignedModulation
  VAR
    lValue : BOOL;
  END_VAR

            ;
          

METHOD test
  VAR_INPUT
    override : BOOL;
  END_VAR
                  IF (override) THEN
	RETURN;
END_IF

clear();

IF (lValue) THEN
	lInterlockState:=cInterlockStateErrorNegative;
	lScalingNegative := 0.0;
	lThresholdNegative := 0.0;
	
	trigger(FALSE);
END_IF

                
END_METHOD

PROPERTY Value : BOOL
GET
                    Value := lValue;
                  
END_GET
SET
                    lValue := Value;
                  
END_SET
END_PROPERTY
END_FUNCTION_BLOCK

FUNCTION_BLOCK ScaledInterlock EXTENDS ReportableSignedModulation
  VAR
    lValue : t_percentage;
    lScalingContext : REFERENCE TO ValueObjectPercentage;
    lScaling : t_percentage;
    lZeroThreshold : t_percentage := 0.05;
  END_VAR

            ;
          

METHOD test
  VAR_INPUT
    override : BOOL;
  END_VAR
                  IF (override) THEN
	RETURN;
END_IF

clear();

IF ((lValue<0) AND (lScalingContext.Value<0) AND (lScaling<>1.0)) THEN
	IF (ABS(lScaling)<ABS(lZeroThreshold)) THEN
		lInterlockState := cInterlockStateErrorNegative;
		lScalingNegative := 0.0;
	ELSE
		lInterlockState := cInterlockStateWarning;
		lScalingNegative := lScaling;
	END_IF
	
	trigger(FALSE);
	RETURN;
END_IF

IF ((lValue>0) AND (lScalingContext.Value>0) AND (lScaling<>1.0)) THEN
	IF (ABS(lScaling)<ABS(lZeroThreshold)) THEN
		lInterlockState  :=cInterlockStateErrorPositive;
		lScalingPositive := 0.0;
	ELSE
		lInterlockState := cInterlockStateWarning;
		lScalingPositive := lScaling;
	END_IF
	
	trigger(FALSE);
	RETURN;
END_IF


                
END_METHOD

PROPERTY Scaling : t_percentage
GET
                    Scaling := lScaling;
                  
END_GET
SET
                    lScaling := Scaling;
                  
END_SET
END_PROPERTY

PROPERTY ScalingContext : REFERENCE TO ValueObjectPercentage
GET
                    ScalingContext ref= lScalingContext;
                  
END_GET
SET
                    lScalingContext ref= ScalingContext;
                  
END_SET
END_PROPERTY

PROPERTY Value : t_percentage
GET
                    Value := lValue;
                  
END_GET
SET
                    lValue := Value;
                  
END_SET
END_PROPERTY

PROPERTY ZeroThreshold : t_percentage
GET
                    ZeroThreshold := lZeroThreshold;
                  
END_GET
SET
                    lZeroThreshold := ZeroThreshold;
                  
END_SET
END_PROPERTY
END_FUNCTION_BLOCK

FUNCTION_BLOCK ThresholdInterlock EXTENDS ReportableSignedModulation
  VAR
    lValue : REAL;
    lThreshold : REAL;
    lTimer : t_timer;
  END_VAR

            ;
          

METHOD initializeState
  VAR_INPUT
    p : POINTER TO t_particle_nop;
    nme : t_token_string;
    code : t_state_code;
  END_VAR
                  SUPER^.initializeState(p,nme,code);

lTimer.initialize();
lTimer.Enable := TRUE;

                
END_METHOD

METHOD test
  VAR_INPUT
    override : BOOL;
  END_VAR
                  lTimer.operator();

IF (override) THEN
	RETURN;
END_IF

clear();

IF (lValue>lThreshold) THEN
	IF (lTimer.Expired) THEN
		lInterlockState:=cInterlockStateError;
		lScalingPositive := 0.0;
		lThresholdPositive := 0.0;
		lScalingNegative := 0.0;
		lThresholdNegative := 0.0;

		trigger(FALSE);
	END_IF
ELSE
	lTimer.reset();
END_IF

                
END_METHOD

PROPERTY Period : t_time
GET
                    Period := lTimer.Period;
                  
END_GET
SET
                    lTimer.Period := Period;
                  
END_SET
END_PROPERTY

PROPERTY Threshold : REAL
GET
                    Threshold := lThreshold;
                  
END_GET
SET
                    lThreshold := Threshold;
                  
END_SET
END_PROPERTY

PROPERTY Value : REAL
GET
                    Value := lValue;
                  
END_GET
SET
                    lValue := Value;
                  
END_SET
END_PROPERTY
END_FUNCTION_BLOCK

FUNCTION_BLOCK SynchronousInterlock EXTENDS NonOperationalParticleSet
  VAR CONSTANT
    cInnerRegion : t_percentage := 0.005;
    cOuterRegion : t_percentage := 0.04;
    cInnerValue : t_percentage := 1.0;
    cOuterValue : t_percentage := 0.0;
    cOuterRegionRelaxed : t_percentage := 0.1;
    cInnerRegionRelaxed : t_percentage := 0.05;
    cInnerValueRelaxed : t_percentage := 1.0;
    cOuterValueRelaxed : t_percentage := 0.0;
    cZeroThreshold : t_percentage := 0.03;
  END_VAR
  VAR
    lClientA : ScaledInterlock;
    lClientB : ScaledInterlock;
    lInputA : REFERENCE TO ValueObjectPercentage;
    lInputB : REFERENCE TO ValueObjectPercentage;
    lForceRelaxed : BOOL := FALSE;
    lSignA : t_percentage := 1.0;
    lSignB : t_percentage := 1.0;
    lTransform : TransformIsoscelesTrapezoid;
    lDelta : t_percentage := 0;
    lAverage : ValueObjectPercentage;
    lScaling : t_percentage;
  END_VAR

            ;
          

METHOD initialize
                  lClientA.initializeState(NopSelf,'',cCCSynchronousInterlock);
lClientB.initializeState(NopSelf,'',cCCSynchronousInterlock);

lTransform.InnerRegion := cInnerRegion;
lTransform.OuterRegion := cOuterRegion;
lTransform.InnerValue := cInnerValue;
lTransform.OuterValue := cOuterValue;

ClientA.ZeroThreshold := cZeroThreshold;
ClientB.ZeroThreshold := cZeroThreshold;

SUPER^.initialize();

                
END_METHOD

METHOD operator
                  lDelta := lInputA.Value - lInputB.Value;

lAverage.Value := (lInputA.Value + lInputB.Value)/2.0;
lAverage.operator();

lScaling := lTransform.compute(lDelta);

lClientA.Value := lDelta * lSignA;
lClientA.Scaling := lScaling;
lClientA.test(FALSE);

lClientB.Value := lDelta * lSignB;
lClientB.Scaling := lScaling;
lClientB.test(FALSE);

SUPER^.operator();

IF (lForceRelaxed) THEN
	relax();
END_IF

                
END_METHOD

METHOD relax
                  lTransform.InnerRegion := cInnerRegionRelaxed;
lTransform.OuterRegion := cOuterRegionRelaxed;
lTransform.InnerValue := cInnerValueRelaxed;
lTransform.OuterValue := cOuterValueRelaxed;

                
END_METHOD

METHOD tighten
                  lTransform.InnerRegion := cInnerRegion;
lTransform.OuterRegion := cOuterRegion;
lTransform.InnerValue := cInnerValue;
lTransform.OuterValue := cOuterValue;

                
END_METHOD

(* {attribute 'monitoring' := 'call'} *)
PROPERTY Average : t_percentage
GET
                    Average := lAverage.Value;
                  
END_GET
END_PROPERTY

PROPERTY AverageObject : REFERENCE TO ValueObjectPercentage
GET
                    AverageObject ref= lAverage;
                  
END_GET
END_PROPERTY

PROPERTY ClientA : REFERENCE TO ScaledInterlock
GET
                    ClientA ref= lClientA;
                  
END_GET
END_PROPERTY

PROPERTY ClientB : REFERENCE TO ScaledInterlock
GET
                    ClientB ref= lClientB;
                  
END_GET
END_PROPERTY

(* {attribute 'monitoring' := 'call'} *)
PROPERTY Delta : t_percentage
GET
                    Delta := lDelta;
                  
END_GET
END_PROPERTY

PROPERTY InputA : REFERENCE TO ValueObjectPercentage
GET
                    InputA ref= lInputA;
                  
END_GET
SET
                    lInputA ref= InputA;
                  
END_SET
END_PROPERTY

PROPERTY InputB : REFERENCE TO ValueObjectPercentage
GET
                    InputB ref= lInputB;
                  
END_GET
SET
                    lInputB ref= InputB;
                  
END_SET
END_PROPERTY

PROPERTY SignA : t_percentage
GET
                    SignA := lSignA;
                  
END_GET
SET
                    lSignA := SignA;
                  
END_SET
END_PROPERTY

PROPERTY SignB : t_percentage
GET
                    SignB := lSignB;
                  
END_GET
SET
                    lSignB := SignB;
                  
END_SET
END_PROPERTY

PROPERTY TypeToken : t_medium_string
GET
                    TypeToken := 'iSynch';
                  
END_GET
END_PROPERTY

PROPERTY ForceRelaxed : BOOL
GET
                    ForceRelaxed := lForceRelaxed;
                  
END_GET
SET
                    lForceRelaxed := ForceRelaxed;
                  
END_SET
END_PROPERTY
END_FUNCTION_BLOCK

FUNCTION_BLOCK WrapperLockoutInterlock EXTENDS NonOperationalParticleSet
  VAR
    lClient : LockoutInterlock;
    lInput : ValueObjectBool;
  END_VAR

            ;
          

METHOD initialize
                  lClient.initializeState(NopSelf,'',cCCLockoutInterlock);

SUPER^.initialize();



                
END_METHOD

METHOD operator
                  lClient.Value := lInput.Value;
lClient.test(FALSE);

SUPER^.operator();

                
END_METHOD

PROPERTY Client : REFERENCE TO LockoutInterlock
GET
                    Client ref= lClient;
                  
END_GET
END_PROPERTY

PROPERTY TypeToken : t_medium_string
GET
                    TypeToken := 'iwLockout';
                  
END_GET
END_PROPERTY
END_FUNCTION_BLOCK

FUNCTION_BLOCK WrapperPositiveOnlyInterlock EXTENDS NonOperationalParticleSet
  VAR
    lClient : PositiveOnlyInterlock;
    lInput : REFERENCE TO ValueObjectBool;
  END_VAR

            ;
          

METHOD initialize
                  lClient.initializeState(NopSelf,'',cCCPosOnlyInterlock);

SUPER^.initialize();


                
END_METHOD

METHOD operator
                  lClient.Value := lInput.Value;
lClient.test(FALSE);

SUPER^.operator();

                
END_METHOD

PROPERTY Client : REFERENCE TO PositiveOnlyInterlock
GET
                    Client ref= lClient;
                  
END_GET
END_PROPERTY

PROPERTY Input : REFERENCE TO ValueObjectBool
GET
                    Input ref= lInput;
                  
END_GET
SET
                    lInput ref= Input;
                  
END_SET
END_PROPERTY

PROPERTY TypeToken : t_medium_string
GET
                    TypeToken := 'iwPosOnly';
                  
END_GET
END_PROPERTY
END_FUNCTION_BLOCK

FUNCTION_BLOCK WrapperScaledInterlock EXTENDS NonOperationalParticleSet
  VAR CONSTANT
    cOuterRegion : t_percentage := 1.0;
    cInnerRegion : t_percentage := 0.7;
    cInnerValue : t_percentage := 1.0;
    cOuterValue : t_percentage := 0.0;
    cZeroThreshold : t_percentage := 0.03;
  END_VAR
  VAR
    lClient : ScaledInterlock;
    lInput : REFERENCE TO ValueObjectPercentage;
    lTransform : TransformIsoscelesTrapezoid;
    lSign : t_percentage := 1.0;
  END_VAR

            ;
          

METHOD initialize
                  lClient.initializeState(NopSelf,'',cCCScaledInterlock);

lTransform.InnerRegion := cInnerRegion;
lTransform.OuterRegion := cOuterRegion;
lTransform.InnerValue := cInnerValue;
lTransform.OuterValue := cOuterValue;

Client.ZeroThreshold := cZeroThreshold;

SUPER^.initialize();

                
END_METHOD

METHOD operator
                  lClient.Value := lInput.Value * lSign;
lClient.Scaling := lTransform.compute(lInput.Value);
lClient.test(FALSE);

SUPER^.operator();

                
END_METHOD

PROPERTY Client : REFERENCE TO ScaledInterlock
GET
                    Client ref= lClient;
                  
END_GET
END_PROPERTY

PROPERTY Input : REFERENCE TO ValueObjectPercentage
GET
                    Input ref= lInput;
                  
END_GET
SET
                    lInput ref= Input;
                  
END_SET
END_PROPERTY

PROPERTY Sign : t_percentage
GET
                    Sign := lSign;
                  
END_GET
SET
                    lSign := Sign;
                  
END_SET
END_PROPERTY

PROPERTY TypeToken : t_medium_string
GET
                    TypeToken := 'iwScaled';
                  
END_GET
END_PROPERTY

PROPERTY Transform : REFERENCE TO TransformIsoscelesTrapezoid
GET
                    Transform ref= lTransform;
                  
END_GET
END_PROPERTY
END_FUNCTION_BLOCK

FUNCTION_BLOCK WrapperThresholdInterlock EXTENDS NonOperationalParticleSet
  VAR
    lClient : ThresholdInterlock;
    lInput : REFERENCE TO ValueObjectReal;
  END_VAR

            ;
          

METHOD initialize
                  lClient.initializeState(NopSelf,'',cCCThresholdInterlock);

SUPER^.initialize();

                
END_METHOD

METHOD operator
                  lClient.Value := lInput.Value;
lClient.test(FALSE);

SUPER^.operator();

                
END_METHOD

PROPERTY Client : REFERENCE TO ThresholdInterlock
GET
                    Client ref= lClient;
                  
END_GET
END_PROPERTY

PROPERTY Input : REFERENCE TO ValueObjectReal
GET
                    Input ref= lInput;
                  
END_GET
SET
                    lInput ref= Input;
                  
END_SET
END_PROPERTY

PROPERTY TypeToken : t_medium_string
GET
                    TypeToken := 'iwThreshold';
                  
END_GET
END_PROPERTY
END_FUNCTION_BLOCK

FUNCTION_BLOCK ChargeEnergyMetric EXTENDS StatisticMetric
  VAR
    _Statistic : SimpleStatistic;
    lCumulativeEnergyCurrent : REAL;
    lCumulativeEnergyPrevious : REAL;
  END_VAR

            ;
          

METHOD initialize
                  Statistic REF= _Statistic;

SUPER^.initialize();

                
END_METHOD

METHOD operator
                  lCumulativeEnergyCurrent := gSystem.lBMS.ChargeCumulativeEnergy;
                
END_METHOD

METHOD start
                  lCumulativeEnergyPrevious := gSystem.lBMS.ChargeCumulativeEnergy;
                
END_METHOD

METHOD stop
                  lValue := lCumulativeEnergyCurrent - lCumulativeEnergyPrevious;

SUPER^.stop();

                
END_METHOD
END_FUNCTION_BLOCK

FUNCTION_BLOCK DischargeEnergyMetric EXTENDS StatisticMetric
  VAR
    _Statistic : SimpleStatistic;
    lCumulativeEnergyCurrent : REAL;
    lCumulativeEnergyPrevious : REAL;
  END_VAR

            ;
          

METHOD initialize
                  Statistic REF= _Statistic;

SUPER^.initialize();

                
END_METHOD

METHOD operator
                  lCumulativeEnergyCurrent := gSystem.lBMS.DischargeCumulativeEnergy;
                
END_METHOD

METHOD start
                  lCumulativeEnergyPrevious := gSystem.lBMS.DischargeCumulativeEnergy;
                
END_METHOD

METHOD stop
                  lValue := lCumulativeEnergyCurrent - lCumulativeEnergyPrevious;

SUPER^.stop();

                
END_METHOD
END_FUNCTION_BLOCK

FUNCTION_BLOCK EnergyMetricSet EXTENDS MetricSet
  VAR
    lChargeEnergyMetric : ChargeEnergyMetric;
    lDischargeEnergyMetric : DischargeEnergyMetric;
  END_VAR

            ;
          

METHOD initialize
                  register(ADR(lChargeEnergyMetric));
register(ADR(lDischargeEnergyMetric));

SUPER^.initialize();

                
END_METHOD
END_FUNCTION_BLOCK

FUNCTION_BLOCK Metric

            ;
          

METHOD cycle
                  stop();
start();

                
END_METHOD

METHOD initialize
                  
                
END_METHOD

METHOD operator
                  
                
END_METHOD

METHOD reset
                  

                
END_METHOD

METHOD start
                  
                
END_METHOD

METHOD stop
                  
                
END_METHOD
END_FUNCTION_BLOCK

FUNCTION_BLOCK MetricSet EXTENDS Metric
  VAR
    lMetricCount : USINT := 0;
    lMetricSet : t_metric_set;
  END_VAR

            
          

METHOD cycle
  VAR
    i : USINT;
  END_VAR
                  FOR i:=1 TO lMetricCount DO
	lMetricSet[i]^.cycle();
END_FOR

                
END_METHOD

METHOD initialize
  VAR
    i : USINT;
  END_VAR
                  FOR i:=1 TO lMetricCount DO
	lMetricSet[i]^.initialize();
END_FOR
                
END_METHOD

METHOD operator
  VAR
    i : USINT;
  END_VAR
                  FOR i:=1 TO lMetricCount DO
	lMetricSet[i]^.operator();
END_FOR
                
END_METHOD

METHOD registerMetric
  VAR_INPUT
    metric : t_metric_ptr;
  END_VAR
                  IF (metric=0) THEN
	RETURN;
END_IF

IF (lMetricCount>=8) THEN
	gCodeErrorHandler(pMessage:='Metric register overflow');
	RETURN;
END_IF

lMetricCount := lMetricCount + 1;
lMetricSet[lMetricCount] := metric;
                
END_METHOD

METHOD reset
  VAR
    i : USINT;
  END_VAR
                  FOR i:=1 TO lMetricCount DO
	lMetricSet[i]^.reset();
END_FOR
                
END_METHOD

METHOD start
  VAR
    i : USINT;
  END_VAR
                  FOR i:=1 TO lMetricCount DO
	lMetricSet[i]^.start();
END_FOR
                
END_METHOD

METHOD stop
  VAR
    i : USINT;
  END_VAR
                  FOR i:=1 TO lMetricCount DO
	lMetricSet[i]^.stop();
END_FOR
                
END_METHOD
END_FUNCTION_BLOCK

FUNCTION_BLOCK EnergyMetric EXTENDS Particle
  VAR_GLOBAL
    sEnergyMetric : t_medium_string := 'EnergyMetric';
  END_VAR
  VAR
    lPower : REAL;
    lCycleEnergy : REAL;
    lCycleTime : REAL;  (* in seconds *)
    lCumulativeEnergy : REAL;
    lTimeStampPrevious : ULINT;
    lTimeStampCurrent : ULINT;
  END_VAR

            ;
          

METHOD initialize
                  SUPER^.initialize();

lPower := 0;
lCycleEnergy := 0;
lCycleTime := 0;
lCumulativeEnergy := 0;

lTimeStampPrevious := 0;
lTimeStampCurrent := 0;


                
END_METHOD

METHOD integrate
  VAR_INPUT
    current : REAL;
    voltage : REAL;
  END_VAR
                  lTimeStampPrevious := lTimeStampCurrent;
lTimeStampCurrent := System.Cycle.SystemTimeMicroseconds;

IF (lTimeStampPrevious=0) THEN
	RETURN;
END_IF

lPower := (current * voltage);
lCycleTime := (ULINT_TO_REAL(lTimeStampCurrent)-ULINT_TO_REAL(lTimeStampPrevious))/1000000.0;
lCycleEnergy := lPower* lCycleTime;
lCumulativeEnergy := lCumulativeEnergy + lCycleEnergy;

                
END_METHOD

METHOD reset
                  lPower := 0;
lCycleEnergy := 0;
lCycleTime := 0;
lCumulativeEnergy := 0;

lTimeStampPrevious := System.Cycle.SystemTimeMicroseconds;
lTimeStampCurrent := System.Cycle.SystemTimeMicroseconds;

// foobar make a command
                
END_METHOD
END_FUNCTION_BLOCK

FUNCTION_BLOCK StatisticMetric EXTENDS Metric
  VAR
    lStatistic : REFERENCE TO Statistic;
    lValue : REAL;
  END_VAR

            ;
          

METHOD initialize
                  SUPER^.initialize();

lStatistic.initialize();

                
END_METHOD

METHOD reset
                  lStatistic.reset();
                
END_METHOD

METHOD stop
                  lStatistic.sample(lValue);
                
END_METHOD
END_FUNCTION_BLOCK

FUNCTION_BLOCK SystemMirror EXTENDS OperationalParticleSet
  VAR
    lExternalState : REFERENCE TO UINT;
    lSupplementaryCommand : REFERENCE TO USINT;
    lInternalState : REFERENCE TO USINT;
    lAlarm : REFERENCE TO USINT;
    lMessage : REFERENCE TO USINT;
    lHealthState : REFERENCE TO UINT;
    lHealthAlarm : REFERENCE TO USINT;
    lHealthTrace : REFERENCE TO USINT;
    lSupplementaryState : REFERENCE TO USINT;
    lSystemState : t_system_state;
    lOperatingMode : t_operating_mode;
    lUMFSAllow : BOOL;
    lGlobalOverride : BOOL;
    lResetDiagnostics : BOOL;
    lResetHardware : BOOL;
    lResetHealth : BOOL;
    lOperatingModeLockRequest : ValueObjectBoolInputReferenceUSINT;
    lOperatingModeRunningRegister : ValueObjectBoolInputReferenceUSINT;
    lUMFSRegister : ValueObjectBoolInputReferenceUSINT;
    lValidTransmissions : ValueObjectBoolInputReferenceUSINT;
    lTPDO1Stuffing : ValueObjectBoolInputReferenceUSINT;
  END_VAR

            ;
          

METHOD initialize
                  IF ((NOT(__ISVALIDREF(lExternalState))) OR
	(NOT(__ISVALIDREF(lSupplementaryCommand))) OR
	(NOT(__ISVALIDREF(lInternalState))) OR
	(NOT(__ISVALIDREF(lAlarm))) OR
	(NOT(__ISVALIDREF(lMessage))) OR
	(NOT(__ISVALIDREF(lHealthState))) OR
	(NOT(__ISVALIDREF(lHealthAlarm))) OR
	(NOT(__ISVALIDREF(lHealthTrace))) OR
	(NOT(__ISVALIDREF(lSupplementaryState)))) THEN
	gCodeErrorHandler(pMessage:=CONCAT('null reference in ',lIdentity));
END_IF

lOperatingModeLockRequest.initializeValueObjectOp(OpSelf,'LockReq','Lock operating mode requested','',cValueStyleConfigurable);
lOperatingModeLockRequest.Index := 0;
lOperatingModeLockRequest.InputReference REF= lInternalState;

lOperatingModeRunningRegister.initializeValueObjectOp(OpSelf,'RunningReg','Running operating mode requested','',cValueStyleConfigurable);
lOperatingModeRunningRegister.Index := 1;
lOperatingModeRunningRegister.InputReference REF= lInternalState;

lUMFSRegister.initializeValueObjectOp(OpSelf,'UMFSReg','UMFS registration requested','',cValueStyleConfigurable);
lUMFSRegister.Index := 2;
lUMFSRegister.InputReference REF= lInternalState;

lValidTransmissions.initializeValueObjectOp(OpSelf,'ValidTrnsmssns','Valid transmissions detected','',cValueStyleConfigurable);
lValidTransmissions.Index := 3;
lValidTransmissions.InputReference REF= lInternalState;

lTPDO1Stuffing.initializeValueObjectOp(OpSelf,'TPDO1Stuffing','TPDO1 stuffing bit detected','',cValueStyleConfigurable);
lTPDO1Stuffing.Index := 7;
lTPDO1Stuffing.InputReference REF= lInternalState;

SUPER^.initialize();
                
END_METHOD

METHOD initializeMirror
  VAR_INPUT
    externalState : REFERENCE TO UINT;
    supplementaryCommand : REFERENCE TO USINT;
    internalState : REFERENCE TO USINT;
    alarm : REFERENCE TO USINT;
    message : REFERENCE TO USINT;
    healthState : REFERENCE TO UINT;
    healthAlarm : REFERENCE TO USINT;
    healthTrace : REFERENCE TO USINT;
    supplementaryState : REFERENCE TO USINT;
  END_VAR
                  lExternalState REF= externalState;
lSupplementaryCommand REF= supplementaryCommand;

lInternalState REF= internalState;
lAlarm REF= alarm;
lMessage REF= message;

lHealthState REF= healthState;
lHealthAlarm REF= healthAlarm;
lHealthTrace REF= healthTrace;

lSupplementaryState REF= supplementaryState;




                
END_METHOD

METHOD operator
                  SUPER^.operator();

lExternalState := 0;
lExternalState := fMergeBitsIntoWord(pWord:=lExternalState,pData:=lSystemState,pStart:=0);
lExternalState := fMergeBitsIntoWord(pWord:=lExternalState,pData:=lOperatingMode,pStart:=4);
lExternalState := fMergeBoolIntoWord(pWord:=lExternalState,pData:=lUMFSAllow,pStart:=8);
lExternalState := fMergeBoolIntoWord(pWord:=lExternalState,pData:=lResetDiagnostics,pStart:=9);
lExternalState := fMergeBoolIntoWord(pWord:=lExternalState,pData:=lResetHardware,pStart:=10);
lExternalState := fMergeBoolIntoWord(pWord:=lExternalState,pData:=lResetHealth,pStart:=11);
lExternalState := fMergeBoolIntoWord(pWord:=lExternalState,pData:=lGlobalOverride,pStart:=12);


                
END_METHOD
END_FUNCTION_BLOCK

FUNCTION_BLOCK SystemMirrorPassThrough EXTENDS SystemMirror
  VAR
    lExternalStateTarget : REFERENCE TO UINT;
    lSupplementaryCommandTarget : REFERENCE TO USINT;
    lInternalStateTarget : REFERENCE TO USINT;
    lAlarmTarget : REFERENCE TO USINT;
    lMessageTarget : REFERENCE TO USINT;
    lHealthStateTarget : REFERENCE TO UINT;
    lHealthAlarmTarget : REFERENCE TO USINT;
    lHealthTraceTarget : REFERENCE TO USINT;
    lSupplementaryStateTarget : REFERENCE TO USINT;
  END_VAR

            ;
          

METHOD initializePassThrough
  VAR_INPUT
    externalState : REFERENCE TO UINT;
    supplementaryCommand : REFERENCE TO USINT;
    internalState : REFERENCE TO USINT;
    alarm : REFERENCE TO USINT;
    message : REFERENCE TO USINT;
    healthState : REFERENCE TO UINT;
    healthAlarm : REFERENCE TO USINT;
    healthTrace : REFERENCE TO USINT;
    supplementaryState : REFERENCE TO USINT;
  END_VAR
                  lExternalStateTarget REF= externalState;
lSupplementaryCommandTarget REF= supplementaryCommand;

lInternalStateTarget REF= internalState;
lAlarmTarget REF= alarm;
lMessageTarget REF= message;

lHealthStateTarget REF= healthState;
lHealthAlarmTarget REF= healthAlarm;
lHealthTraceTarget REF= healthTrace;

lSupplementaryStateTarget REF= supplementaryState;



                
END_METHOD

METHOD operator
                  SUPER^.operator();

(* traffic FROM master PLC *)

lExternalState := lExternalStateTarget;
lSupplementaryCommand := lSupplementaryCommandTarget;
	
(* traffic to master PLC *)

lInternalStateTarget := lInternalState;
lAlarmTarget := lAlarm;
lMessageTarget := lMessage;

lHealthStateTarget := lHealthState;
lHealthAlarmTarget := lHealthAlarm;
lHealthTraceTarget := lHealthTrace;

lSupplementaryStateTarget := lSupplementaryState;
                
END_METHOD

METHOD initialize
                  IF ((NOT(__ISVALIDREF(lExternalStateTarget))) OR
	(NOT(__ISVALIDREF(lSupplementaryCommandTarget))) OR
	(NOT(__ISVALIDREF(lInternalStateTarget))) OR
	(NOT(__ISVALIDREF(lAlarmTarget))) OR
	(NOT(__ISVALIDREF(lMessageTarget))) OR
	(NOT(__ISVALIDREF(lHealthStateTarget))) OR
	(NOT(__ISVALIDREF(lHealthAlarmTarget))) OR
	(NOT(__ISVALIDREF(lHealthTraceTarget))) OR
	(NOT(__ISVALIDREF(lSupplementaryStateTarget)))) THEN
	gCodeErrorHandler(pMessage:=CONCAT('null reference in ',lIdentity));
END_IF

SUPER^.initialize();
                
END_METHOD
END_FUNCTION_BLOCK

FUNCTION_BLOCK OutputSystemState EXTENDS OperationalParticleSet
  VAR
    lVRTriggerCycleOutput : ValueReferenceBool;
    lTriggerCycleOutput : BOOL := FALSE;
    lCausalCycleOutput : ReportableCausal;
    lCycleOutputTimer : t_timer;
    lCycleOutputValue : BOOL := FALSE;
    lOutput : ValueObjectBoolOutputReferenceDINTAsBoolOpt;
    lOutputSystemState : t_system_state := cSystemStateOperational;
  END_VAR

            ;
          

METHOD initialize
                  lVRTriggerCycleOutput.initializeValueReference(lTriggerCycleOutput,NopSelf,'CycleOutput','Power cycle the output','',cValueStyleParameter);

lCausalCycleOutput.initializeState(NopSelf,'',cCCCycleOutput);

lOutput.initializeValueObjectOp(OpSelf,'Output','The output of the object','',cValueStyleConfigurable);

SUPER^.initialize();

lCycleOutputTimer.Enable := TRUE;
lCycleOutputTimer.Period := T#1000MS;
lCycleOutputTimer.initialize();
                
END_METHOD

METHOD off
                  lOutput.off();
                
END_METHOD

METHOD on
                  IF (gSystemServices.SystemState.State<lOutputSystemState) THEN
	RETURN;
END_IF

lOutput.on();

                
END_METHOD

METHOD operator
                  IF (lTriggerCycleOutput) THEN
	lTriggerCycleOutput := FALSE;
	cycleOutput();
END_IF

lCycleOutputTimer.operator();
IF (NOT(lCycleOutputTimer.Expired)) THEN
	lOutput.Value := lCycleOutputValue;
END_IF

IF (gSystemServices.SystemState.State<lOutputSystemState) THEN
	lOutput.off();
END_IF

lOutput.operator();

SUPER^.operator();

                
END_METHOD

METHOD toggleOutput
                  IF (gSystemServices.SystemState.State<lOutputSystemState) THEN
	RETURN;
END_IF

lOutput.Value := NOT(lOutput.Value);

                
END_METHOD

METHOD initializeOutput
  VAR_INPUT
    output : REFERENCE TO DINT;
  END_VAR
                  lOutput.OutputReference ref= output;
                
END_METHOD

METHOD cycleOutput
                  IF (gSystemServices.SystemState.State<lOutputSystemState) THEN
	RETURN;
END_IF

lCycleOutputTimer.reset();
lCycleOutputValue := NOT(lOutput.Value);
lOutput.Value := lCycleOutputValue;

lCausalCycleOutput.trigger(FALSE);

                
END_METHOD

PROPERTY OK : BOOL
GET
                    OK := (lOutput.Value);
                  
END_GET
END_PROPERTY

PROPERTY OutputObject : REFERENCE TO ValueObjectBoolOutputReferenceDINTAsBoolOpt
GET
                    OutputObject ref= lOutput;
                  
END_GET
END_PROPERTY

PROPERTY OutputSystemState : t_system_state
GET
                    OutputSystemState := lOutputSystemState;
                  
END_GET
SET
                    lOutputSystemState := OutputSystemState;
                  
END_SET
END_PROPERTY

PROPERTY TypeToken : t_medium_string
GET
                    TypeToken := 'oSystemState';
                  
END_GET
END_PROPERTY

PROPERTY State : BOOL
GET
                    State := lOutput.Value;
                  
END_GET
END_PROPERTY

PROPERTY Period : t_time
GET
                    Period := lCycleOutputTimer.Period;
                  
END_GET
SET
                    lCycleOutputTimer.Period := Period;
                  
END_SET
END_PROPERTY
END_FUNCTION_BLOCK

FUNCTION_BLOCK OutputSystemStateAuto EXTENDS OutputSystemState

            ;
          

METHOD operator
                  lOutput.Value := (gSystemServices.SystemState.State>=lOutputSystemState);

SUPER^.operator();


                
END_METHOD

METHOD cycleOutput
                  IF (gSystemServices.SystemState.State<lOutputSystemState) THEN
	RETURN;
END_IF

lCycleOutputTimer.reset();
lCycleOutputValue := FALSE;
lOutput.Value := FALSE;

lCausalCycleOutput.trigger(FALSE);

                
END_METHOD

PROPERTY TypeToken : t_medium_string
GET
                    TypeToken := 'oSysStateAuto';
                  
END_GET
END_PROPERTY
END_FUNCTION_BLOCK

FUNCTION_BLOCK OutputSystemStateTimedOn EXTENDS OutputSystemState

            ;
          

METHOD cycleOutput
                  IF (gSystemServices.SystemState.State<lOutputSystemState) THEN
	RETURN;
END_IF

lCycleOutputTimer.reset();
lCycleOutputValue := TRUE;
lOutput.Value := TRUE;

lCausalCycleOutput.trigger(FALSE);

                
END_METHOD

METHOD initialize
                  SUPER^.initialize();

Period := T#5S;

                
END_METHOD

PROPERTY TypeToken : t_medium_string
GET
                    TypeToken := 'oSysStateTimedOn';
                  
END_GET
END_PROPERTY
END_FUNCTION_BLOCK

FUNCTION_BLOCK PackChannel
  VAR
    lPackerSet : t_packer_set;
    lPackerCount : USINT := 0;
    lIndex : USINT := 1;
  END_VAR

            
          

METHOD trigger : BOOL
  VAR_INPUT
    packet : REFERENCE TO t_packet;
    machineStateId : t_machine_state_id;
  END_VAR
  VAR
    i : USINT;
  END_VAR
                  FOR i:=1 TO lPackerCount DO
	IF (lPackerSet[i]^.trigger(packet,machineStateId)) THEN
		RETURN;
	END_IF
END_FOR

                
END_METHOD

METHOD pack
  VAR_INPUT
    packet : REFERENCE TO t_packet;
  END_VAR
                  CurrentPacker.pack(packet);
next();


                
END_METHOD

METHOD initialize
  VAR
    i : USINT;
  END_VAR
                  IF (lPackerCount=0) THEN
	gCodeErrorHandler(pMessage:='empty PackChannel');
END_IF

lIndex := 1;

FOR i:=1 TO lPackerCount DO
	lPackerSet[i]^.initialize();
END_FOR

                
END_METHOD

METHOD unpack
  VAR_INPUT
    packet : REFERENCE TO t_packet;
  END_VAR
  VAR
    i : USINT;
  END_VAR
                  CurrentCode := packet.Code;
CurrentPacker.unpack(packet);


                
END_METHOD

METHOD operator
                  


                
END_METHOD

METHOD register
  VAR_INPUT
    packer : POINTER TO t_packer;
  END_VAR
                  IF (packer=0) THEN
	RETURN;
END_IF

IF (lPackerCount>=16) THEN
	RETURN;
END_IF

lPackerCount := lPackerCount + 1;
lPackerSet[lPackerCount] := packer;
                
END_METHOD

METHOD next
  VAR
    i : USINT;
  END_VAR
                  increment();

i:= 0;
WHILE (NOT(lPackerSet[lIndex]^.Enable)) DO
	increment();
	i := i+1;
	
	IF (i>lPackerCount) THEN
		lIndex := 0;
		RETURN;
	END_IF
END_WHILE

                
END_METHOD

METHOD increment
                  lIndex := lIndex + 1;
IF (lIndex>lPackerCount) THEN
	lIndex := MIN(lPackerCount,1);
END_IF

                
END_METHOD

PROPERTY CurrentPacker : REFERENCE TO t_packer
GET
                    CurrentPacker ref= lPackerSet[lIndex]^;
                  
END_GET
END_PROPERTY

PROPERTY CurrentCode : USINT
GET
                    CurrentCode := CurrentPacker.Code;
                  
END_GET
SET
  VAR
    i : USINT;
  END_VAR
                    IF (CurrentPacker.Code=CurrentCode) THEN
	RETURN;
END_IF

// matches request to Code if possible (Code is present and enabled) otherwise defaults to first regardless of whether it is enabled
FOR i:=1 TO lPackerCount DO
	IF ((lPackerSet[i]^.Code=CurrentCode) AND (lPackerSet[i]^.Enable)) THEN
		lIndex := i;
		RETURN;
	END_IF
END_FOR

// assumes always at least one packer in the channel
lIndex := 1;
                  
END_SET
END_PROPERTY
END_FUNCTION_BLOCK

FUNCTION_BLOCK Packer
  VAR
    lEnable : BOOL := TRUE;
    lCode : USINT := 0;
  END_VAR

            
          

METHOD reset
                  
                
END_METHOD

METHOD unpack
  VAR_INPUT
    packet : REFERENCE TO t_packet;
  END_VAR
                  IF (NOT(lEnable)) THEN
	RETURN;
END_IF

_unpack(packet);
write();
reset();

                
END_METHOD

METHOD _pack
  VAR_INPUT
    packet : REFERENCE TO t_packet;
  END_VAR
                  
                
END_METHOD

METHOD pack
  VAR_INPUT
    packet : REFERENCE TO t_packet;
  END_VAR
                  IF (NOT(lEnable)) THEN
	RETURN;
END_IF

packet.clear();
packet.Code := lCode;

read();
_pack(packet);
reset();

                
END_METHOD

METHOD initialize
                  ;
                
END_METHOD

METHOD _unpack
  VAR_INPUT
    packet : REFERENCE TO t_packet;
  END_VAR
                  
                
END_METHOD

METHOD trigger : BOOL
  VAR_INPUT
    packet : REFERENCE TO t_packet;
    machineStateId : t_machine_state_id;
  END_VAR
                  trigger := FALSE;

                
END_METHOD

METHOD read
                  
                
END_METHOD

METHOD write
                  
                
END_METHOD

PROPERTY Enable : BOOL
GET
                    Enable := lEnable;
                  
END_GET
SET
                    lEnable := Enable;
                  
END_SET
END_PROPERTY

PROPERTY Code : USINT
GET
                    Code := lCode;
                  
END_GET
END_PROPERTY
END_FUNCTION_BLOCK

FUNCTION_BLOCK PacketCANBus
  VAR
    lBuffer : t_bitarray;
    lLatch : BOOL := FALSE;
    lClear : BOOL := FALSE;
  END_VAR

            
          

METHOD copy
  VAR_INPUT
    source : REFERENCE TO t_packet;
  END_VAR
                  IF (NOT(__ISVALIDREF(source))) THEN
	RETURN;
END_IF

IF (lClear) THEN
	Byte1 := 0;
	Byte2 := 0;
	Byte3 := 0;
	Byte4 := 0;
	Byte5 := 0;
	Byte6 := 0;
	Byte7 := 0;
	Byte8 := 0;
END_IF

IF (lLatch) THEN
	Byte1 := Byte1 OR source.Byte1;
	Byte2 := Byte2 OR source.Byte2;
	Byte3 := Byte3 OR source.Byte3;
	Byte4 := Byte4 OR source.Byte4;
	Byte5 := Byte5 OR source.Byte5;
	Byte6 := Byte6 OR source.Byte6;
	Byte7 := Byte7 OR source.Byte7;
	Byte8 := Byte8 OR source.Byte8;	
ELSE
	Byte1 := source.Byte1;
	Byte2 := source.Byte2;
	Byte3 := source.Byte3;
	Byte4 := source.Byte4;
	Byte5 := source.Byte5;
	Byte6 := source.Byte6;
	Byte7 := source.Byte7;
	Byte8 := source.Byte8;	
END_IF

                
END_METHOD

METHOD packBool
  VAR_INPUT
    data : BOOL;
    index : USINT;
  END_VAR
                  lBuffer[index] := data;

                
END_METHOD

METHOD packSINT
  VAR_INPUT
    data : SINT;
    index : USINT;
    length : USINT;
  END_VAR
  VAR
    i : USINT;
    j : USINT;
  END_VAR
                  j := length - 1;

FOR i:=0 TO j DO
	lBuffer[index] := data.0;
	data := SHR(data,1);
	index := index + 1;
END_FOR
                
END_METHOD

METHOD packUINT
  VAR_INPUT
    data : UINT;
    index : USINT;
    length : USINT;
  END_VAR
  VAR
    i : USINT;
    j : USINT;
  END_VAR
                  j := length - 1;

FOR i:=0 TO j DO
	lBuffer[index] := data.0;
	data := SHR(data,1);
	index := index + 1;
END_FOR
                
END_METHOD

METHOD packUSINT
  VAR_INPUT
    data : USINT;
    index : USINT;
    length : USINT;
  END_VAR
  VAR
    i : USINT;
    j : USINT;
  END_VAR
                  j := length - 1;

FOR i:=0 TO j DO
	lBuffer[index] := data.0;
	data := SHR(data,1);
	index := index + 1;
END_FOR
                
END_METHOD

METHOD unpackBool : BOOL
  VAR_INPUT
    index : USINT;
  END_VAR
                  unpackBool := lBuffer[index];
                
END_METHOD

METHOD unpackSINT : SINT
  VAR_INPUT
    index : USINT;
    length : USINT;
  END_VAR
  VAR
    i : USINT;
    j : USINT;
    data : SINT;
  END_VAR
                  j := length - 1;
data := 0;

FOR i:=0 TO j DO
	data := BYTE_TO_SINT(SINT_TO_BYTE(data) OR (SHL(BOOL_TO_BYTE(lBuffer[index]),i)));
	index := index + 1;
END_FOR

unpackSINT := data;
                
END_METHOD

METHOD unpackUINT : UINT
  VAR_INPUT
    index : USINT;
    length : USINT;
  END_VAR
  VAR
    i : USINT;
    j : USINT;
    data : UINT;
  END_VAR
                  j := length - 1;
data := 0;

FOR i:=0 TO j DO
	data := UINT_TO_WORD(data) OR (SHL(BOOL_TO_WORD(lBuffer[index]),i));
	index := index + 1;
END_FOR

unpackUINT := data;
                
END_METHOD

METHOD unpackUSINT : USINT
  VAR_INPUT
    index : USINT;
    length : USINT;
  END_VAR
  VAR
    i : USINT;
    j : USINT;
    data : USINT;
  END_VAR
                  j := length - 1;
data := 0;

FOR i:=0 TO j DO
	data := USINT_TO_BYTE(data) OR (SHL(BOOL_TO_BYTE(lBuffer[index]),i));
	index := index + 1;
END_FOR

unpackUSINT := data;
                
END_METHOD

METHOD clear
                  MEMUtils.Memset(ADR(lBuffer[1]),0,64);
                
END_METHOD

PROPERTY Byte8 : USINT
GET
                    Byte8.0 := Buffer[57];
Byte8.1 := Buffer[58];
Byte8.2 := Buffer[59];
Byte8.3 := Buffer[60];
Byte8.4 := Buffer[61];
Byte8.5 := Buffer[62];
Byte8.6 := Buffer[63];
Byte8.7 := Buffer[64];
                  
END_GET
SET
                    Buffer[57] := Byte8.0;
Buffer[58] := Byte8.1;
Buffer[59] := Byte8.2;
Buffer[60] := Byte8.3;
Buffer[61] := Byte8.4;
Buffer[62] := Byte8.5;
Buffer[63] := Byte8.6;
Buffer[64] := Byte8.7;

                  
END_SET
END_PROPERTY

PROPERTY Byte7 : USINT
GET
                    Byte7.0 := Buffer[49];
Byte7.1 := Buffer[50];
Byte7.2 := Buffer[51];
Byte7.3 := Buffer[52];
Byte7.4 := Buffer[53];
Byte7.5 := Buffer[54];
Byte7.6 := Buffer[55];
Byte7.7 := Buffer[56];
                  
END_GET
SET
                    Buffer[49] := Byte7.0;
Buffer[50] := Byte7.1;
Buffer[51] := Byte7.2;
Buffer[52] := Byte7.3;
Buffer[53] := Byte7.4;
Buffer[54] := Byte7.5;
Buffer[55] := Byte7.6;
Buffer[56] := Byte7.7;

                  
END_SET
END_PROPERTY

PROPERTY Code : USINT
GET
                    Code := unpackUSINT(1,4);
                  
END_GET
SET
                    packUSINT(INT_TO_USINT(Code),1,4);
                  
END_SET
END_PROPERTY

PROPERTY Buffer : REFERENCE TO t_bitarray
GET
                    Buffer ref= lBuffer;
                  
END_GET
END_PROPERTY

PROPERTY Byte1 : USINT
GET
                    Byte1.0 := Buffer[1];
Byte1.1 := Buffer[2];
Byte1.2 := Buffer[3];
Byte1.3 := Buffer[4];
Byte1.4 := Buffer[5];
Byte1.5 := Buffer[6];
Byte1.6 := Buffer[7];
Byte1.7 := Buffer[8];
                  
END_GET
SET
                    Buffer[1] := Byte1.0;
Buffer[2] := Byte1.1;
Buffer[3] := Byte1.2;
Buffer[4] := Byte1.3;
Buffer[5] := Byte1.4;
Buffer[6] := Byte1.5;
Buffer[7] := Byte1.6;
Buffer[8] := Byte1.7;

                  
END_SET
END_PROPERTY

PROPERTY Byte2 : USINT
GET
                    Byte2.0 := Buffer[9];
Byte2.1 := Buffer[10];
Byte2.2 := Buffer[11];
Byte2.3 := Buffer[12];
Byte2.4 := Buffer[13];
Byte2.5 := Buffer[14];
Byte2.6 := Buffer[15];
Byte2.7 := Buffer[16];
                  
END_GET
SET
                    Buffer[9] := Byte2.0;
Buffer[10] := Byte2.1;
Buffer[11] := Byte2.2;
Buffer[12] := Byte2.3;
Buffer[13] := Byte2.4;
Buffer[14] := Byte2.5;
Buffer[15] := Byte2.6;
Buffer[16] := Byte2.7;

                  
END_SET
END_PROPERTY

PROPERTY Byte3 : USINT
GET
                    Byte3.0 := Buffer[17];
Byte3.1 := Buffer[18];
Byte3.2 := Buffer[19];
Byte3.3 := Buffer[20];
Byte3.4 := Buffer[21];
Byte3.5 := Buffer[22];
Byte3.6 := Buffer[23];
Byte3.7 := Buffer[24];
                  
END_GET
SET
                    Buffer[17] := Byte3.0;
Buffer[18] := Byte3.1;
Buffer[19] := Byte3.2;
Buffer[20] := Byte3.3;
Buffer[21] := Byte3.4;
Buffer[22] := Byte3.5;
Buffer[23] := Byte3.6;
Buffer[24] := Byte3.7;

                  
END_SET
END_PROPERTY

PROPERTY Byte4 : USINT
GET
                    Byte4.0 := Buffer[25];
Byte4.1 := Buffer[26];
Byte4.2 := Buffer[27];
Byte4.3 := Buffer[28];
Byte4.4 := Buffer[29];
Byte4.5 := Buffer[30];
Byte4.6 := Buffer[31];
Byte4.7 := Buffer[32];
                  
END_GET
SET
                    Buffer[25] := Byte4.0;
Buffer[26] := Byte4.1;
Buffer[27] := Byte4.2;
Buffer[28] := Byte4.3;
Buffer[29] := Byte4.4;
Buffer[30] := Byte4.5;
Buffer[31] := Byte4.6;
Buffer[32] := Byte4.7;

                  
END_SET
END_PROPERTY

PROPERTY Byte5 : USINT
GET
                    Byte5.0 := Buffer[33];
Byte5.1 := Buffer[34];
Byte5.2 := Buffer[35];
Byte5.3 := Buffer[36];
Byte5.4 := Buffer[37];
Byte5.5 := Buffer[38];
Byte5.6 := Buffer[39];
Byte5.7 := Buffer[40];
                  
END_GET
SET
                    Buffer[33] := Byte5.0;
Buffer[34] := Byte5.1;
Buffer[35] := Byte5.2;
Buffer[36] := Byte5.3;
Buffer[37] := Byte5.4;
Buffer[38] := Byte5.5;
Buffer[39] := Byte5.6;
Buffer[40] := Byte5.7;

                  
END_SET
END_PROPERTY

PROPERTY Byte6 : USINT
GET
                    Byte6.0 := Buffer[41];
Byte6.1 := Buffer[42];
Byte6.2 := Buffer[43];
Byte6.3 := Buffer[44];
Byte6.4 := Buffer[45];
Byte6.5 := Buffer[46];
Byte6.6 := Buffer[47];
Byte6.7 := Buffer[48];
                  
END_GET
SET
                    Buffer[41] := Byte6.0;
Buffer[42] := Byte6.1;
Buffer[43] := Byte6.2;
Buffer[44] := Byte6.3;
Buffer[45] := Byte6.4;
Buffer[46] := Byte6.5;
Buffer[47] := Byte6.6;
Buffer[48] := Byte6.7;

                  
END_SET
END_PROPERTY
END_FUNCTION_BLOCK

FUNCTION AngleAsSint : SINT
  VAR_INPUT
    lInput : REAL;
  END_VAR
  VAR CONSTANT
    lLowerBound : REAL := cPi;
    lUpperBound : REAL := cPi;
  END_VAR
  VAR
    lValue : REAL;
  END_VAR

            (* lower and upper bounds should be equal *)
IF (lInput>0) THEN
	lValue := MIN(1.0,lInput/lUpperBound)*127.0;
ELSE
	lValue := MAX(-1.0,lInput/lLowerBound)*(128.0);
END_IF

AngleAsSint := REAL_TO_SINT(lValue);
          
END_FUNCTION

FUNCTION AngleAsUsintDeprecated : USINT
  VAR_INPUT
    lInput : REAL;
  END_VAR
  VAR CONSTANT
    lLowerBound : REAL := cPiNegative;
    lUpperBound : REAL := cPi;
  END_VAR

            AngleAsUsintDeprecated := REAL_TO_USINT((MAX(lLowerBound,MIN(lUpperBound,lInput))/(lUpperBound-lLowerBound)*256.0)+128.0);

          
END_FUNCTION

FUNCTION AngleFromSint : REAL
  VAR_INPUT
    lInput : SINT;
  END_VAR
  VAR CONSTANT
    lLowerBound : REAL := cPi;
    lUpperBound : REAL := cPi;
  END_VAR
  VAR
    lValue : REAL;
  END_VAR

            (* lower and upper bounds should be equal *)
IF (lInput>0) THEN
	AngleFromSint := SINT_TO_REAL(lInput)/127.0*lUpperBound;
ELSE
	AngleFromSint := SINT_TO_REAL(lInput)/128*lLowerBound;
END_IF

          
END_FUNCTION

FUNCTION Decode7bitSINT : SINT
  VAR_INPUT
    data : USINT;
  END_VAR

            Decode7bitSINT := INT_TO_SINT(MAX((USINT_TO_INT(data)*2),255)-128);

          
END_FUNCTION

FUNCTION_BLOCK PackArray
  VAR_INPUT
    in : USINT;
    lIndex : BYTE;
    lWidth : BYTE;
    lRef : REFERENCE TO t_bitarray;
  END_VAR
  VAR_OUTPUT
    out : USINT;
  END_VAR

            
          

ACTION initialize:
                
              
END_ACTION

METHOD pack : BOOL
  VAR_INPUT
    data : USINT;
  END_VAR
                  packBoolArray(data:=data,
	ref:=lRef,
	index:=lIndex,
	width:=lWidth);
	
pack := TRUE;
                
END_METHOD

METHOD unpack : USINT
                  unpack := unpackBoolArray(
	ref:=lRef,
	index:=lIndex,
	width:=lWidth);
                
END_METHOD
END_FUNCTION_BLOCK

FUNCTION_BLOCK PackArray1
  VAR_INPUT
    in : BOOL;
    lIndex : BYTE;
    lRef : REFERENCE TO t_bitarray;
  END_VAR
  VAR_OUTPUT
    out : BOOL;
  END_VAR

            
          

ACTION initialize:
                
              
END_ACTION

METHOD pack : BOOL
  VAR_INPUT
    data : BOOL;
  END_VAR
                  packBoolArray(data:=BOOL_TO_USINT(data),
	ref:=lRef,
	index:=lIndex,
	width:=1);
	
pack := TRUE;
                
END_METHOD

METHOD unpack : BOOL
                  unpack := USINT_TO_BOOL(unpackBoolArray(
	ref:=lRef,
	index:=lIndex,
	width:=1));
	
                
END_METHOD
END_FUNCTION_BLOCK

FUNCTION_BLOCK PackArray16
  VAR_INPUT
    in : UINT;
    lIndex : BYTE;
    lRef : REFERENCE TO t_bitarray;
  END_VAR
  VAR_OUTPUT
    out : UINT;
  END_VAR

            
          

ACTION initialize:
                
              
END_ACTION

METHOD pack : BOOL
  VAR_INPUT
    data : UINT;
  END_VAR
                  packBoolArray16(data:=data,
	ref:=lRef,
	index:=lIndex,
	width:=16);
	
pack := TRUE;
                
END_METHOD

METHOD unpack : UINT
                  unpack := unpackBoolArray16(
	ref:=lRef,
	index:=lIndex,
	width:=16);
                
END_METHOD
END_FUNCTION_BLOCK

FUNCTION_BLOCK PackArray8
  VAR_INPUT
    in : USINT;
    lIndex : BYTE;
    lRef : REFERENCE TO t_bitarray;
  END_VAR
  VAR_OUTPUT
    out : USINT;
  END_VAR

            
          

ACTION initialize:
                
              
END_ACTION

METHOD pack : BOOL
  VAR_INPUT
    data : USINT;
  END_VAR
                  packBoolArray(data:=data,
	ref:=lRef,
	index:=lIndex,
	width:=8);
	
pack := TRUE;
                
END_METHOD

METHOD unpack : USINT
                  unpack := unpackBoolArray(
	ref:=lRef,
	index:=lIndex,
	width:=8);
                
END_METHOD
END_FUNCTION_BLOCK

FUNCTION packBoolArray : BOOL
  VAR_INPUT
    ref : REFERENCE TO t_bitarray;
    index : BYTE;
    width : BYTE;
    data : USINT;
  END_VAR
  VAR
    i : BYTE;
    j : BYTE;
  END_VAR

            packBoolArray := TRUE;

j := width - 1;

FOR i:=0 TO j DO
	ref[index] := data.0;
	data := SHR(data,1);
	index := index + 1;
END_FOR

          
END_FUNCTION

FUNCTION packBoolArray16 : BOOL
  VAR_INPUT
    ref : REFERENCE TO t_bitarray;
    index : BYTE;
    width : BYTE;
    data : UINT;
  END_VAR
  VAR
    i : BYTE;
    j : BYTE;
  END_VAR

            packBoolArray16 := TRUE;

j := width - 1;

FOR i:=0 TO j DO
	ref[index] := data.0;
	data := SHR(data,1);
	index := index + 1;
END_FOR


          
END_FUNCTION

FUNCTION PercentageAs4bits : USINT
  VAR_INPUT
    lInput : t_percentage;
  END_VAR

            PercentageAs4bits := REAL_TO_USINT(MAX(0.0,MIN(15.0/16.0,ABS(lInput)))*16);
          
END_FUNCTION

FUNCTION PercentageAs5bits : USINT
  VAR_INPUT
    lInput : t_percentage;
  END_VAR

            PercentageAs5bits := REAL_TO_USINT(MAX(0.0,MIN(31.0/32.0,ABS(lInput)))*32);
          
END_FUNCTION

FUNCTION PercentageAs7bits : USINT
  VAR_INPUT
    lInput : t_percentage;
  END_VAR

            PercentageAs7bits := REAL_TO_USINT(MAX(0.0,MIN(127.0/128.0,ABS(lInput)))*128);
          
END_FUNCTION

FUNCTION PercentageAsSint : SINT
  VAR_INPUT
    lInput : t_percentage;
  END_VAR
  VAR
    lValue : REAL;
  END_VAR

            IF (lInput>0) THEN
	lValue := MIN(1.0,lInput)*100.0;
ELSE
	lValue := MAX(-1.0,lInput)*100.0;
END_IF

PercentageAsSint := REAL_TO_SINT(lValue);
          
END_FUNCTION

FUNCTION PercentageAsUsintDeprecated : USINT
  VAR_INPUT
    lInput : t_percentage;
  END_VAR
  VAR
    lValue : REAL;
  END_VAR

            IF (lInput>0) THEN
	lValue := MIN(1.0,lInput)*127.0;
ELSE
	lValue := MAX(-1.0,lInput)*128.0;
END_IF

PercentageAsUsintDeprecated := REAL_TO_USINT(lValue+128);

          
END_FUNCTION

FUNCTION PercentageFrom4bits : t_percentage
  VAR_INPUT
    lInput : USINT;
  END_VAR

            PercentageFrom4bits := USINT_TO_REAL(lInput)/16.0;
          
END_FUNCTION

FUNCTION PercentageFrom5bits : t_percentage
  VAR_INPUT
    lInput : USINT;
  END_VAR

            PercentageFrom5bits := USINT_TO_REAL(lInput)/32.0;
          
END_FUNCTION

FUNCTION PercentageFrom7bits : t_percentage
  VAR_INPUT
    lInput : USINT;
  END_VAR

            PercentageFrom7bits := USINT_TO_REAL(lInput)/128.0;
          
END_FUNCTION

FUNCTION SignedPercentageAs5bits : USINT
  VAR_INPUT
    lInput : t_percentage;
  END_VAR

            SignedPercentageAs5bits := REAL_TO_USINT((MAX(-1.0,MIN(15.0/16.0,lInput))+1.0)*16);
          
END_FUNCTION

FUNCTION SignedPercentageAs6bits : USINT
  VAR_INPUT
    lInput : t_percentage;
  END_VAR

            SignedPercentageAs6bits := REAL_TO_USINT((MAX(-1.0,MIN(31.0/32.0,lInput))+1.0)*32);
          
END_FUNCTION

FUNCTION SignedPercentageAs7bits : USINT
  VAR_INPUT
    lInput : t_percentage;
  END_VAR

            SignedPercentageAs7bits := REAL_TO_USINT((MAX(-1.0,MIN(63.0/64.0,lInput))+1.0)*64);
          
END_FUNCTION

FUNCTION SignedPercentageAs8bits : USINT
  VAR_INPUT
    lInput : t_percentage;
  END_VAR

            SignedPercentageAs8bits := REAL_TO_USINT((MAX(-1.0,MIN(127.0/128.0,lInput))+1.0)*128);
          
END_FUNCTION

FUNCTION SignedPercentageFrom5bits : t_percentage
  VAR_INPUT
    lInput : USINT;
  END_VAR

            SignedPercentageFrom5bits := USINT_TO_REAL(lInput)/16.0 - 1.0;

          
END_FUNCTION

FUNCTION SignedPercentageFrom6bits : t_percentage
  VAR_INPUT
    lInput : USINT;
  END_VAR

            SignedPercentageFrom6bits := USINT_TO_REAL(lInput)/32.0 - 1.0;

          
END_FUNCTION

FUNCTION SignedPercentageFrom7bits : t_percentage
  VAR_INPUT
    lInput : USINT;
  END_VAR

            SignedPercentageFrom7bits := USINT_TO_REAL(lInput)/64.0 - 1.0;

          
END_FUNCTION

FUNCTION SignedPercentageFrom8bits : t_percentage
  VAR_INPUT
    lInput : USINT;
  END_VAR

            SignedPercentageFrom8bits := USINT_TO_REAL(lInput)/128.0 - 1.0;

          
END_FUNCTION

FUNCTION unpackBoolArray : USINT
  VAR_INPUT
    ref : REFERENCE TO t_bitarray;
    index : BYTE;
    width : BYTE;
  END_VAR
  VAR
    data : USINT := 0;
    i : BYTE;
    j : BYTE;
  END_VAR

            j := width - 1;

FOR i:=0 TO j DO
	data := USINT_TO_BYTE(data) OR (SHL(BOOL_TO_BYTE(ref[index]),i));
	index := index + 1;
END_FOR

unpackBoolArray := data;
          
END_FUNCTION

FUNCTION unpackBoolArray16 : UINT
  VAR_INPUT
    ref : REFERENCE TO t_bitarray;
    index : BYTE;
    width : BYTE;
  END_VAR
  VAR
    data : UINT := 0;
    i : BYTE;
    j : BYTE;
  END_VAR

            j := width - 1;

FOR i:=0 TO j DO
	data := UINT_TO_WORD(data) OR (SHL(BOOL_TO_WORD(ref[index]),i));
	index := index + 1;
END_FOR

unpackBoolArray16 := data;
          
END_FUNCTION

FUNCTION_BLOCK SecondaryPowerSupply EXTENDS NonOperationalParticleSet
  VAR CONSTANT
    cSecondaryTargetVoltage : REAL := 13.0;
  END_VAR
  VAR_GLOBAL
    sSecondaryPowerSupply : t_medium_string := 'Secondary';
  END_VAR
  VAR
    lAlarmSecondaryWaiting : ReportableAlarmAllowableUp;
    lAlarmSecondaryNotRunning : ReportableAlarmEscalating;
    lAlarmSecondaryNotRunningModulation : ReportableSignedModulation;
    lAlarmRunStateMismatch : ReportableAlarmEscalating;
    lModulation : ReportableContextSignedModulation;
    lAvailability : t_percentage;
    lModulationSeverity : t_severity;
    lRequestedState : t_run_state;
    lCurrentState : t_run_state;
    lTargetVoltage : REAL;
    lControllerSecondaryPowerSupplyA : REFERENCE TO ControllerSecondaryPowerSupply;
    lControllerSecondaryPowerSupplyB : REFERENCE TO ControllerSecondaryPowerSupply;
  END_VAR

            ;
          

METHOD initialize
                  IF ((NOT(__ISVALIDREF(lControllerSecondaryPowerSupplyA))) OR
	(NOT(__ISVALIDREF(lControllerSecondaryPowerSupplyB)))) THEN
	gCodeErrorHandler(pMessage:=CONCAT('null reference in ',lIdentity));
END_IF

lAlarmSecondaryNotRunning.initializeState(NopSelf,'',cACSecondaryNotRunning); // foobar escalates to pause
lAlarmSecondaryNotRunning.Life := 10;
lAlarmSecondaryNotRunning.InitialSeverity := cSeverityNone;
lAlarmSecondaryNotRunning.SeverityWarningTimeout := T#1S;
lAlarmSecondaryNotRunning.SeverityErrorTimeout := T#2S;
lAlarmSecondaryNotRunning.SeverityCriticalTimeout := T#5S;

lAlarmSecondaryNotRunningModulation.initializeState(NopSelf,'',cACSecondaryNotRunningModulation); // foobar life was zero
lAlarmSecondaryNotRunningModulation.pause();
lAlarmSecondaryNotRunningModulation.registerServer(ADR(lModulation));

lAlarmSecondaryWaiting.initializeState(NopSelf,'',cACSecondaryWaiting);
lAlarmSecondaryWaiting.AllowableSystemState := cSystemStatePreparing;
lAlarmSecondaryWaiting.UpperSystemStateScope := cSystemStatePreparing;
lAlarmSecondaryWaiting.LowerSystemStateScope := cSystemStatePreparing;
lAlarmSecondaryWaiting.Life := 10;
lAlarmSecondaryWaiting.InitialSeverity := cSeverityNone;
lAlarmSecondaryWaiting.SeverityWarningTimeout := T#1S;
lAlarmSecondaryWaiting.SeverityErrorTimeout := T#2S;
lAlarmSecondaryWaiting.SeverityCriticalTimeout := T#5S;

lAlarmRunStateMismatch.initializeState(NopSelf,'',cACSecondaryRunStateMismatch);
lAlarmRunStateMismatch.InitialSeverity := cSeverityNone;
lAlarmRunStateMismatch.SeverityWarningTimeout := T#1S;
lAlarmRunStateMismatch.SeverityErrorTimeout := T#2S;
lAlarmRunStateMismatch.SeverityCriticalTimeout := T#5S;

lModulation.initializeEvent(NopSelf,'',cECSecondaryPowerModulation);

SUPER^.initialize();
SubSystem := cSubsystemSecondary;

lModulationSeverity := cSeverityError;
lTargetVoltage := cSecondaryTargetVoltage;
                
END_METHOD

METHOD operator
                  lCurrentState := cRunStateNone;

IF ((lControllerSecondaryPowerSupplyA.CurrentRunState=cRunStateStop) OR
	(lControllerSecondaryPowerSupplyA.CurrentRunState=cRunStateStop)) THEN
	lCurrentState := cRunStateStop;
END_IF

IF ((lControllerSecondaryPowerSupplyA.CurrentRunState=cRunStateStart) OR
	(lControllerSecondaryPowerSupplyA.CurrentRunState=cRunStateStart)) THEN
	lCurrentState := cRunStateStart;
END_IF
	
IF (lControllerSecondaryPowerSupplyA.CurrentRunState<>lControllerSecondaryPowerSupplyB.CurrentRunState) THEN
	lAlarmRunStateMismatch.trigger(FALSE); // foobar any further action
END_IF

SUPER^.operator();

lRequestedState := cRunStateStop;
lAvailability := 0.0;

IF (gSystemServices.SystemState.State<cSystemStatePreparing) THEN
	RETURN;
END_IF

IF (BMSConnected) THEN
	lRequestedState := cRunStateStart;
END_IF

IF (lCurrentState<>cRunStateStart) THEN
	lAlarmSecondaryNotRunning.trigger(FALSE);
	
	IF (lAlarmSecondaryNotRunning.Severity>=lModulationSeverity) THEN
		lAlarmSecondaryNotRunningModulation.trigger(FALSE);
	END_IF

	lAlarmSecondaryWaiting.test(FALSE);	
END_IF

lModulation.operator();
lAvailability := MIN(lModulation.ScalingPositive,lModulation.ThresholdPositive);

lControllerSecondaryPowerSupplyA.RequestedRunState := lRequestedState;
lControllerSecondaryPowerSupplyB.RequestedRunState := lRequestedState;

lControllerSecondaryPowerSupplyA.TargetVoltage := lTargetVoltage;
lControllerSecondaryPowerSupplyB.TargetVoltage := lTargetVoltage;

                
END_METHOD
END_FUNCTION_BLOCK

FUNCTION_BLOCK SecondaryPowerSupplyPrimary EXTENDS SecondaryPowerSupply

            ;
          

METHOD initialize
                  SUPER^.initialize();

lControllerSecondaryPowerSupplyA REF= gSystem.lCANOpenMasterSystem.SecondaryPowerSupplyA;
lControllerSecondaryPowerSupplyB REF= gSystem.lCANOpenMasterSystem.SecondaryPowerSupplyB;

                
END_METHOD
END_FUNCTION_BLOCK

FUNCTION_BLOCK Active EXTENDS OperationalParticleSet
  VAR CONSTANT
    cActivePreTimeout : t_time := TIME#0ms;
    cActivePostTimeout : t_time := TIME#0ms;
  END_VAR
  VAR
    lAllow : ValueObjectBool;
    lPreTimer : t_timer;
    lPostTimer : t_timer;
    lState : t_active_state := t_active_state.cActiveStateNone;
    lRegisterActive : BOOL := FALSE;
    lValue : BOOL := FALSE;
    lAllowPreCondition : BOOL := TRUE;
  END_VAR

            ;
          

METHOD active
                  IF (NOT(lValue)) THEN
	lPostTimer.reset();
	lState := t_active_state.cActiveStatePost;
END_IF
                
END_METHOD

METHOD inactive
                  IF (lValue) THEN
	lPreTimer.reset();
	lState := t_active_state.cActiveStatePre;
	transitionOutOfInactive();
END_IF
                
END_METHOD

METHOD initialize
                  lAllow.initializeValueObjectOp(OpSelf,'Allow','Dependent operations are allowed','',cValueStyleConfigurable);

SUPER^.initialize();

lPreTimer.lEnable := TRUE;
lPreTimer.lPeriod := cActivePreTimeout;
lPreTimer.initialize();

lPostTimer.lEnable := TRUE;
lPostTimer.lPeriod := cActivePostTimeout;
lPostTimer.initialize();

lRegisterActive := FALSE;
lValue := FALSE;
lState := t_active_state.cActiveStateNone;

                
END_METHOD

METHOD operator
                  lValue := lRegisterActive;
lRegisterActive := FALSE;

lPreTimer.operator();
lPostTimer.operator();

CASE (lState) OF
	t_active_state.cActiveStateNone:
		inactive();
	t_active_state.cActiveStatePre:
		pre();
	t_active_state.cActiveStatePost:
		post();
	t_active_state.cActiveStateActive:
		active();
END_CASE

IF (gSystemServices.SystemState.State<>cSystemStateOperational) THEN
	lState := t_active_state.cActiveStateNone;
END_IF

lAllow.Value := ((lState>t_active_state.cActiveStatePre) AND (lAllowPreCondition));

SUPER^.operator();

                
END_METHOD

METHOD post
                  IF (lValue) THEN
	lState := t_active_state.cActiveStateActive;
	RETURN;
END_IF

IF (lPostTimer.lExpired) THEN
	lState := t_active_state.cActiveStateNone;
END_IF
                
END_METHOD

METHOD pre
                  IF (NOT(lValue)) THEN
	lState := t_active_state.cActiveStateNone;
	RETURN;
END_IF

IF (lPreTimer.lExpired) THEN
	lState := t_active_state.cActiveStateActive;
END_IF

                
END_METHOD

METHOD registerActive
                  lRegisterActive := TRUE;
                
END_METHOD

METHOD transitionOutOfInactive
                  ;
                
END_METHOD

PROPERTY Allow : BOOL
GET
                    Allow := lAllow.Value;

                  
END_GET
END_PROPERTY

PROPERTY IsActive : BOOL
GET
                    IsActive := (lState<>t_active_state.cActiveStateNone);

                  
END_GET
END_PROPERTY

PROPERTY PostPeriod : t_time
GET
                    PostPeriod := lPostTimer.Period;
                  
END_GET
SET
                    lPostTimer.Period := PostPeriod;
                  
END_SET
END_PROPERTY

PROPERTY PrePeriod : t_time
GET
                    PrePeriod := lPreTimer.Period;
                  
END_GET
SET
                    lPreTimer.Period := PrePeriod;
                  
END_SET
END_PROPERTY

PROPERTY State : t_active_state
GET
                    State := lState;
                  
END_GET
END_PROPERTY

PROPERTY TriggerRegisterActive : BOOL
SET
                    IF (TriggerRegisterActive) THEN
	registerActive();
END_IF
                  
END_SET
END_PROPERTY

PROPERTY TypeToken : t_medium_string
GET
                    TypeToken := 'Active';
                  
END_GET
END_PROPERTY
END_FUNCTION_BLOCK

FUNCTION_BLOCK Cycle EXTENDS OperationalParticleSet
  VAR_GLOBAL
    sDefaultAverageCycleTime : ULINT := 32000;
  END_VAR
  VAR
    lVRTriggerResetStatistics : ValueReferenceBool;
    lTriggerResetStatistics : BOOL := FALSE;
    lVRTriggerResetHours : ValueReferenceBool;
    lTriggerResetHours : BOOL := FALSE;
    lVRTriggerResetOperationalHours : ValueReferenceBool;
    lTriggerResetOperationalHours : BOOL := FALSE;
    lVRTriggerResetStartCount : ValueReferenceBool;
    lTriggerResetStartCount : BOOL := FALSE;
    lCurrentTime : ValueObjectULINTInputReferenceULINT;
    lStartTime : t_persistent_ulint;
    lStartCount : t_persistent_uint;
    lReset : BOOL;
    lFirstCycle : BOOL := TRUE;
    lTimeStep : t_timestep;
    lPreviousStartTime : ULINT;
    lPreviousTime : ULINT;
    lToggleTime : ULINT;
    lSyncClockTickPrevious : ULINT;
    lAverageCycleTime : ULINT := sDefaultAverageCycleTime;
    lAveragingFactor : REAL := 0.9;
    lCycleTime : ULINT := 30000;
    lMinCycleTime : ULINT;
    lMaxCycleTime : ULINT;
    lSystemTIme : t_medium_string;
    lIntegralClockTickPrevious : ULINT;
    lIntegralStartTime : ULINT;
    lIntegralPeriod : ULINT := 1000000;
    lIntegralClockTick : BOOL;
    lIntegralRunning : BOOL := FALSE;
    lIntegralReset : BOOL := FALSE;
    lIntegralDuration : ULINT;
    lCounter : USINT := 0;
    lToggle : BOOL;
    lToggleTransition : BOOL;
    lTogglePeriodMicroseconds : ULINT := 150000;
  END_VAR

            ;
          

METHOD initialize
                  lVRTriggerResetStatistics.initializeValueReference(lTriggerResetStatistics,NopSelf,'ResetStats','Reset all statistics','',cValueStyleTrigger);
lVRTriggerResetHours.initializeValueReference(lTriggerResetHours,NopSelf,'ResetHours','Reset up-time hours','',cValueStyleTrigger);
lVRTriggerResetOperationalHours.initializeValueReference(lTriggerResetOperationalHours,NopSelf,'ResetOpHours','Reset operational hours','',cValueStyleTrigger);
lVRTriggerResetStartCount.initializeValueReference(lTriggerResetStartCount,NopSelf,'ResetStartCnt','Reset plc start count','',cValueStyleTrigger);

lCurrentTime.initializeValueObjectOp(OpSelf,'CurrentTime','Current system time','timestep',cValueStyleConfigurable);

lStartTime.Identifier := t_persistent_id.cPersistentID_StartTimeMicroseconds;
lStartTime.initialize();

lStartCount.Identifier := t_persistent_id.cPersistentID_StartCount;
lStartCount.initialize();

SUPER^.initialize();

lStartCount.Value := lStartCount.Value + 1;

lCurrentTime.operator();

lFirstCycle := TRUE;
lTimeStep := 0;
lPreviousTime := 0;

lIntegralClockTickPrevious := lCurrentTime.Value;
lIntegralClockTick := FALSE;

lCycleTime := sDefaultAverageCycleTime;
lToggleTime := lCurrentTime.Value;

lMaxCycleTime := 0;
lMinCycleTime := 1000000000;

lPreviousStartTime := lStartTime.Value;
lStartTime.Value := lCurrentTime.Value;


                
END_METHOD

METHOD operator
                  lPreviousTime := lCurrentTime.Value;

SUPER^.operator();

IF (lTriggerResetStatistics) THEN
	lTriggerResetStatistics := FALSE;

	lMaxCycleTime := 0;
	lMinCycleTime := 1000000;
END_IF

IF (lTriggerResetHours) THEN
	lTriggerResetHours := FALSE;

	Hours := 0;
END_IF

IF (lTriggerResetOperationalHours) THEN
	lTriggerResetOperationalHours := FALSE;

	OperationalHours := 0;
END_IF
	
IF (lTriggerResetStartCount) THEN
	lTriggerResetStartCount := FALSE;

	lStartCount.Value := 0;
END_IF

lCycleTime := lCurrentTime.Value - lPreviousTime;
IF (NOT(lFirstCycle)) THEN
	lMinCycleTime := MIN(lMinCycleTime,lCycleTime);
	lMaxCycleTime := MAX(lMaxCycleTime,lCycleTime);
	
	lAverageCycleTime := REAL_TO_ULINT(ULINT_TO_REAL(lAverageCycleTime)*0.9 + ULINT_TO_REAL(lCycleTime)*0.1);
END_IF
lFirstCycle := FALSE;
lTimeStep := lTimeStep + 1;

lSystemTime := ULINT_TO_STRING(lTimeStep);

